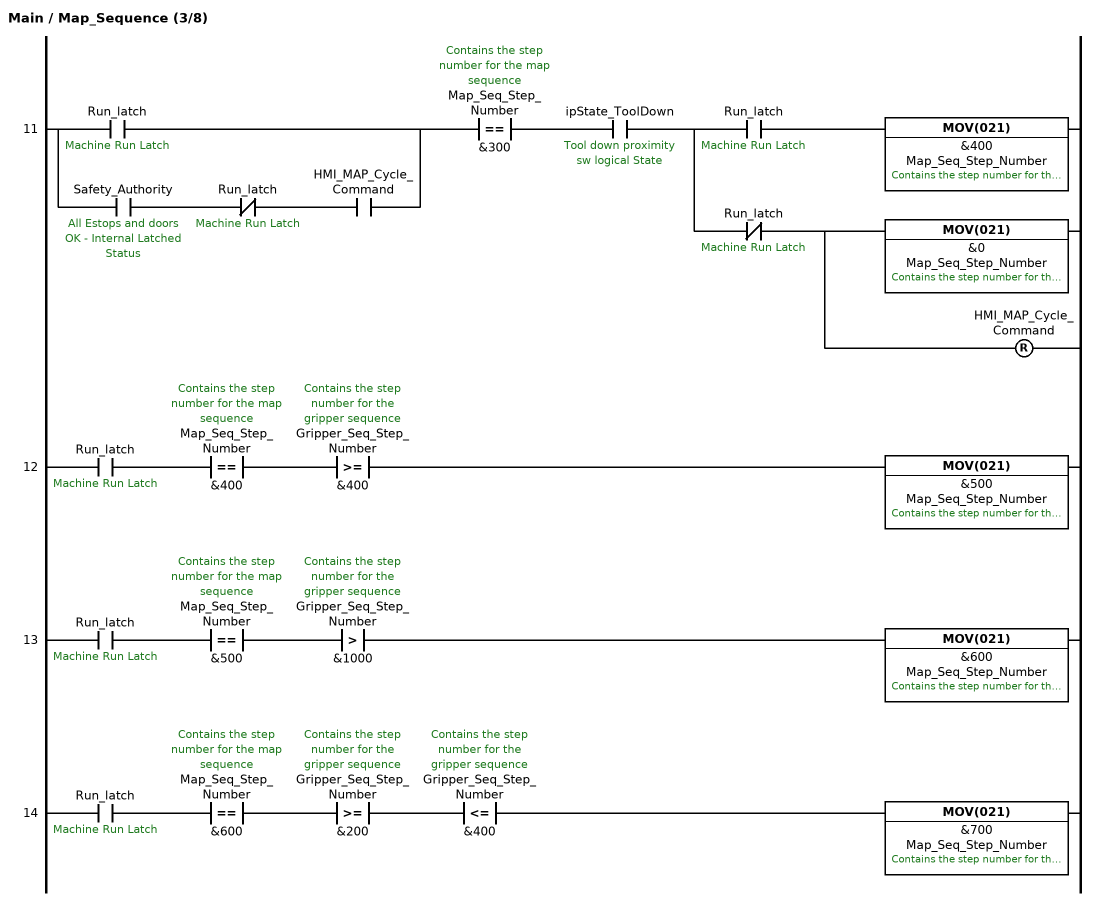
; [picture p48: Main / Map_Sequence, rungs 11-14]
; rung 11
LD Run_latch  ; Machine Run Latch
LD Safety_Authority  ; All Estops and doors OK - Internal Latched Status
ANDNOT Run_latch  ; Machine Run Latch
AND HMI_MAP_Cycle_Command
ORLD
AND=(300) Map_Seq_Step_Number &300  ; Contains the step number for the map sequence
AND ipState_ToolDown  ; Tool down proximity sw logical State
OUT TR0
AND Run_latch  ; Machine Run Latch
MOV(021) &400 Map_Seq_Step_Number  ; Contains the step number for the map sequence
LD TR0
ANDNOT Run_latch  ; Machine Run Latch
MOV(021) &0 Map_Seq_Step_Number  ; Contains the step number for the map sequence
RSET HMI_MAP_Cycle_Command
; rung 12
LD Run_latch  ; Machine Run Latch
AND=(300) Map_Seq_Step_Number &400  ; Contains the step number for the map sequence
AND>=(325) Gripper_Seq_Step_Number &400  ; Contains the step number for the gripper sequence
MOV(021) &500 Map_Seq_Step_Number  ; Contains the step number for the map sequence
; rung 13
LD Run_latch  ; Machine Run Latch
AND=(300) Map_Seq_Step_Number &500  ; Contains the step number for the map sequence
AND>(320) Gripper_Seq_Step_Number &1000  ; Contains the step number for the gripper sequence
MOV(021) &600 Map_Seq_Step_Number  ; Contains the step number for the map sequence
; rung 14
LD Run_latch  ; Machine Run Latch
AND=(300) Map_Seq_Step_Number &600  ; Contains the step number for the map sequence
AND>=(325) Gripper_Seq_Step_Number &200  ; Contains the step number for the gripper sequence
AND<=(315) Gripper_Seq_Step_Number &400  ; Contains the step number for the gripper sequence
MOV(021) &700 Map_Seq_Step_Number  ; Contains the step number for the map sequence

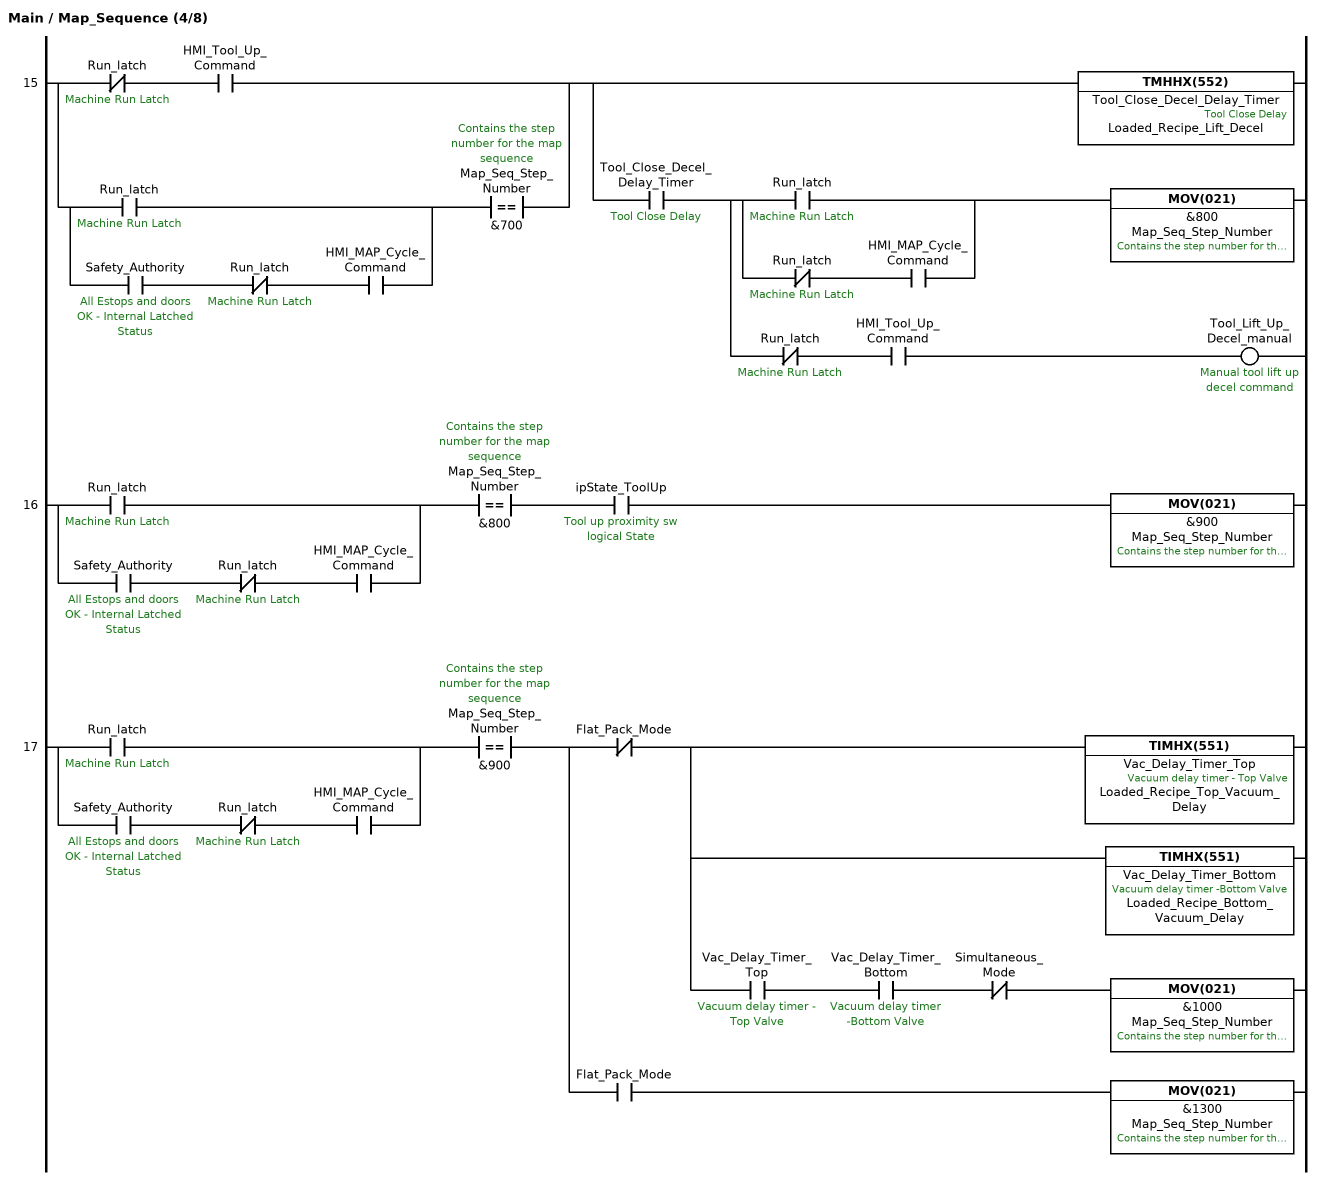
; rung 15
LDNOT Run_latch  ; Machine Run Latch
AND HMI_Tool_Up_Command
LD Run_latch  ; Machine Run Latch
LD Safety_Authority  ; All Estops and doors OK - Internal Latched Status
ANDNOT Run_latch  ; Machine Run Latch
AND HMI_MAP_Cycle_Command
ORLD
AND=(300) Map_Seq_Step_Number &700  ; Contains the step number for the map sequence
ORLD
TMHHX(552) Tool_Close_Decel_Delay_Timer Loaded_Recipe_Lift_Decel  ; Tool Close Delay
AND Tool_Close_Decel_Delay_Timer  ; Tool Close Delay
OUT TR0
LD Run_latch  ; Machine Run Latch
LDNOT Run_latch  ; Machine Run Latch
AND HMI_MAP_Cycle_Command
ORLD
ANDLD
MOV(021) &800 Map_Seq_Step_Number  ; Contains the step number for the map sequence
LD TR0
ANDNOT Run_latch  ; Machine Run Latch
AND HMI_Tool_Up_Command
OUT Tool_Lift_Up_Decel_manual  ; Manual tool lift up decel command
; rung 16
LD Run_latch  ; Machine Run Latch
LD Safety_Authority  ; All Estops and doors OK - Internal Latched Status
ANDNOT Run_latch  ; Machine Run Latch
AND HMI_MAP_Cycle_Command
ORLD
AND=(300) Map_Seq_Step_Number &800  ; Contains the step number for the map sequence
AND ipState_ToolUp  ; Tool up proximity sw logical State
MOV(021) &900 Map_Seq_Step_Number  ; Contains the step number for the map sequence
; rung 17
LD Run_latch  ; Machine Run Latch
LD Safety_Authority  ; All Estops and doors OK - Internal Latched Status
ANDNOT Run_latch  ; Machine Run Latch
AND HMI_MAP_Cycle_Command
ORLD
AND=(300) Map_Seq_Step_Number &900  ; Contains the step number for the map sequence
OUT TR0
ANDNOT Flat_Pack_Mode
TIMHX(551) Vac_Delay_Timer_Top Loaded_Recipe_Top_Vacuum_Delay  ; Vacuum delay timer - Top Valve
TIMHX(551) Vac_Delay_Timer_Bottom Loaded_Recipe_Bottom_Vacuum_Delay  ; Vacuum delay timer -Bottom Valve
AND Vac_Delay_Timer_Top  ; Vacuum delay timer - Top Valve
AND Vac_Delay_Timer_Bottom  ; Vacuum delay timer -Bottom Valve
ANDNOT Simultaneous_Mode
MOV(021) &1000 Map_Seq_Step_Number  ; Contains the step number for the map sequence
LD TR0
AND Flat_Pack_Mode
MOV(021) &1300 Map_Seq_Step_Number  ; Contains the step number for the map sequence

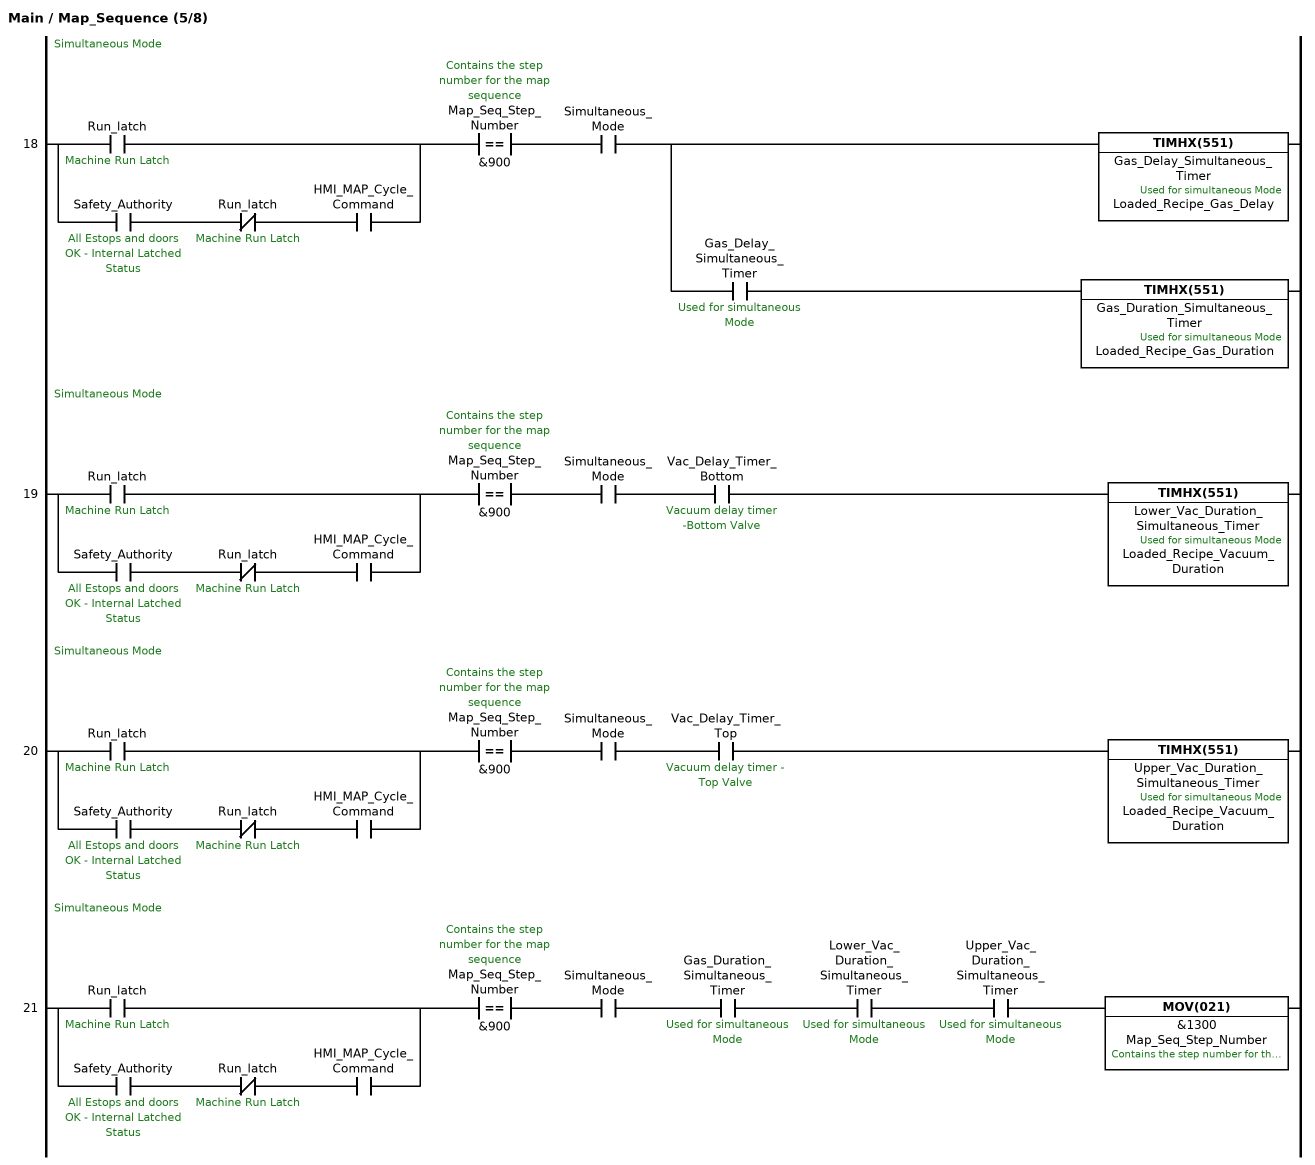
; rung 18: Simultaneous Mode
LD Run_latch  ; Machine Run Latch
LD Safety_Authority  ; All Estops and doors OK - Internal Latched Status
ANDNOT Run_latch  ; Machine Run Latch
AND HMI_MAP_Cycle_Command
ORLD
AND=(300) Map_Seq_Step_Number &900  ; Contains the step number for the map sequence
AND Simultaneous_Mode
TIMHX(551) Gas_Delay_Simultaneous_Timer Loaded_Recipe_Gas_Delay  ; Used for simultaneous Mode
AND Gas_Delay_Simultaneous_Timer  ; Used for simultaneous Mode
TIMHX(551) Gas_Duration_Simultaneous_Timer Loaded_Recipe_Gas_Duration  ; Used for simultaneous Mode
; rung 19: Simultaneous Mode
LD Run_latch  ; Machine Run Latch
LD Safety_Authority  ; All Estops and doors OK - Internal Latched Status
ANDNOT Run_latch  ; Machine Run Latch
AND HMI_MAP_Cycle_Command
ORLD
AND=(300) Map_Seq_Step_Number &900  ; Contains the step number for the map sequence
AND Simultaneous_Mode
AND Vac_Delay_Timer_Bottom  ; Vacuum delay timer -Bottom Valve
TIMHX(551) Lower_Vac_Duration_Simultaneous_Timer Loaded_Recipe_Vacuum_Duration  ; Used for simultaneous Mode
; rung 20: Simultaneous Mode
LD Run_latch  ; Machine Run Latch
LD Safety_Authority  ; All Estops and doors OK - Internal Latched Status
ANDNOT Run_latch  ; Machine Run Latch
AND HMI_MAP_Cycle_Command
ORLD
AND=(300) Map_Seq_Step_Number &900  ; Contains the step number for the map sequence
AND Simultaneous_Mode
AND Vac_Delay_Timer_Top  ; Vacuum delay timer - Top Valve
TIMHX(551) Upper_Vac_Duration_Simultaneous_Timer Loaded_Recipe_Vacuum_Duration  ; Used for simultaneous Mode
; rung 21: Simultaneous Mode
LD Run_latch  ; Machine Run Latch
LD Safety_Authority  ; All Estops and doors OK - Internal Latched Status
ANDNOT Run_latch  ; Machine Run Latch
AND HMI_MAP_Cycle_Command
ORLD
AND=(300) Map_Seq_Step_Number &900  ; Contains the step number for the map sequence
AND Simultaneous_Mode
AND Gas_Duration_Simultaneous_Timer  ; Used for simultaneous Mode
AND Lower_Vac_Duration_Simultaneous_Timer  ; Used for simultaneous Mode
AND Upper_Vac_Duration_Simultaneous_Timer  ; Used for simultaneous Mode
MOV(021) &1300 Map_Seq_Step_Number  ; Contains the step number for the map sequence

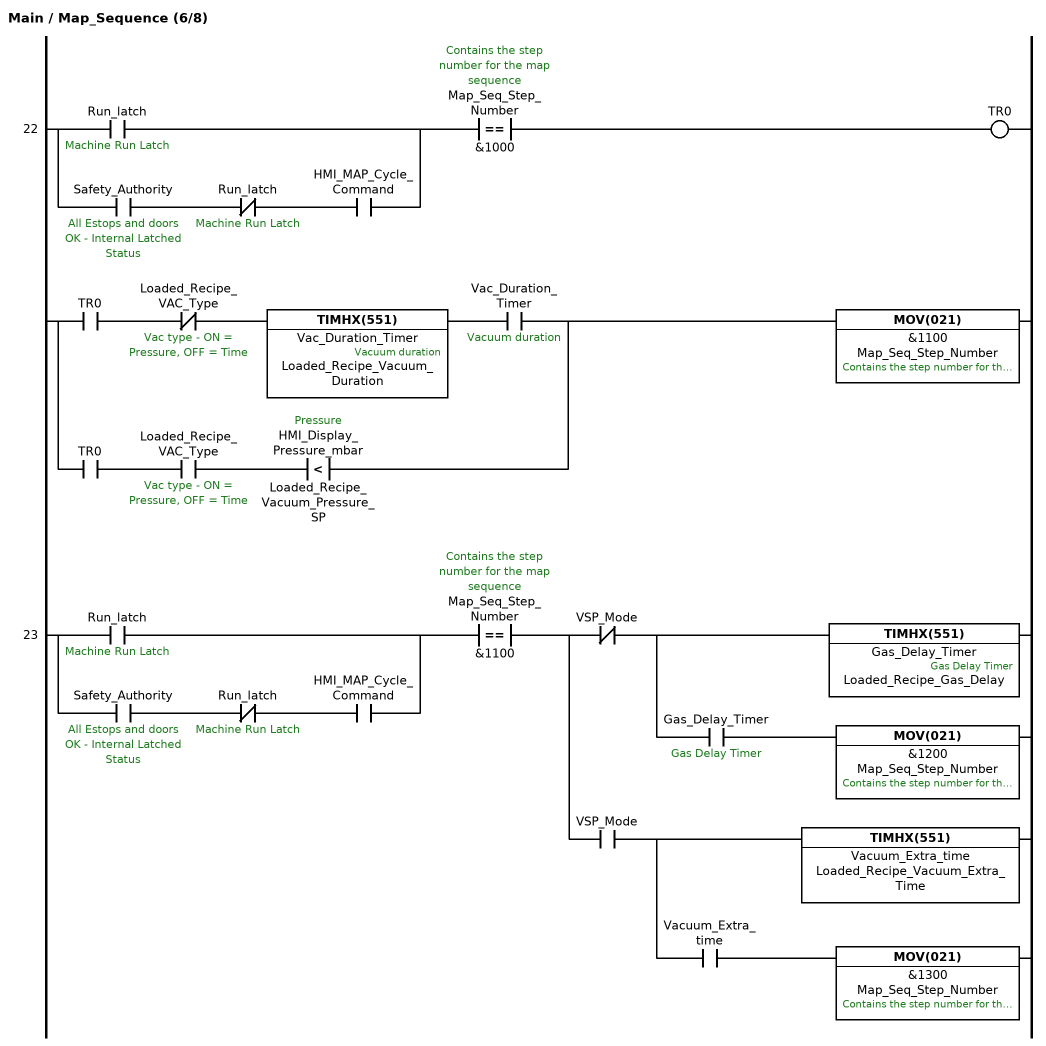
; rung 22
LD Run_latch  ; Machine Run Latch
LD Safety_Authority  ; All Estops and doors OK - Internal Latched Status
ANDNOT Run_latch  ; Machine Run Latch
AND HMI_MAP_Cycle_Command
ORLD
AND=(300) Map_Seq_Step_Number &1000  ; Contains the step number for the map sequence
OUT TR0
ANDNOT Loaded_Recipe_VAC_Type  ; Vac type - ON = Pressure, OFF = Time
TIMHX(551) Vac_Duration_Timer Loaded_Recipe_Vacuum_Duration  ; Vacuum duration
AND Vac_Duration_Timer  ; Vacuum duration
LD TR0
AND Loaded_Recipe_VAC_Type  ; Vac type - ON = Pressure, OFF = Time
AND<(310) HMI_Display_Pressure_mbar Loaded_Recipe_Vacuum_Pressure_SP  ; Pressure
ORLD
MOV(021) &1100 Map_Seq_Step_Number  ; Contains the step number for the map sequence
; rung 23
LD Run_latch  ; Machine Run Latch
LD Safety_Authority  ; All Estops and doors OK - Internal Latched Status
ANDNOT Run_latch  ; Machine Run Latch
AND HMI_MAP_Cycle_Command
ORLD
AND=(300) Map_Seq_Step_Number &1100  ; Contains the step number for the map sequence
OUT TR0
ANDNOT VSP_Mode
TIMHX(551) Gas_Delay_Timer Loaded_Recipe_Gas_Delay  ; Gas Delay Timer
AND Gas_Delay_Timer  ; Gas Delay Timer
MOV(021) &1200 Map_Seq_Step_Number  ; Contains the step number for the map sequence
LD TR0
AND VSP_Mode
TIMHX(551) Vacuum_Extra_time Loaded_Recipe_Vacuum_Extra_Time
AND Vacuum_Extra_time
MOV(021) &1300 Map_Seq_Step_Number  ; Contains the step number for the map sequence

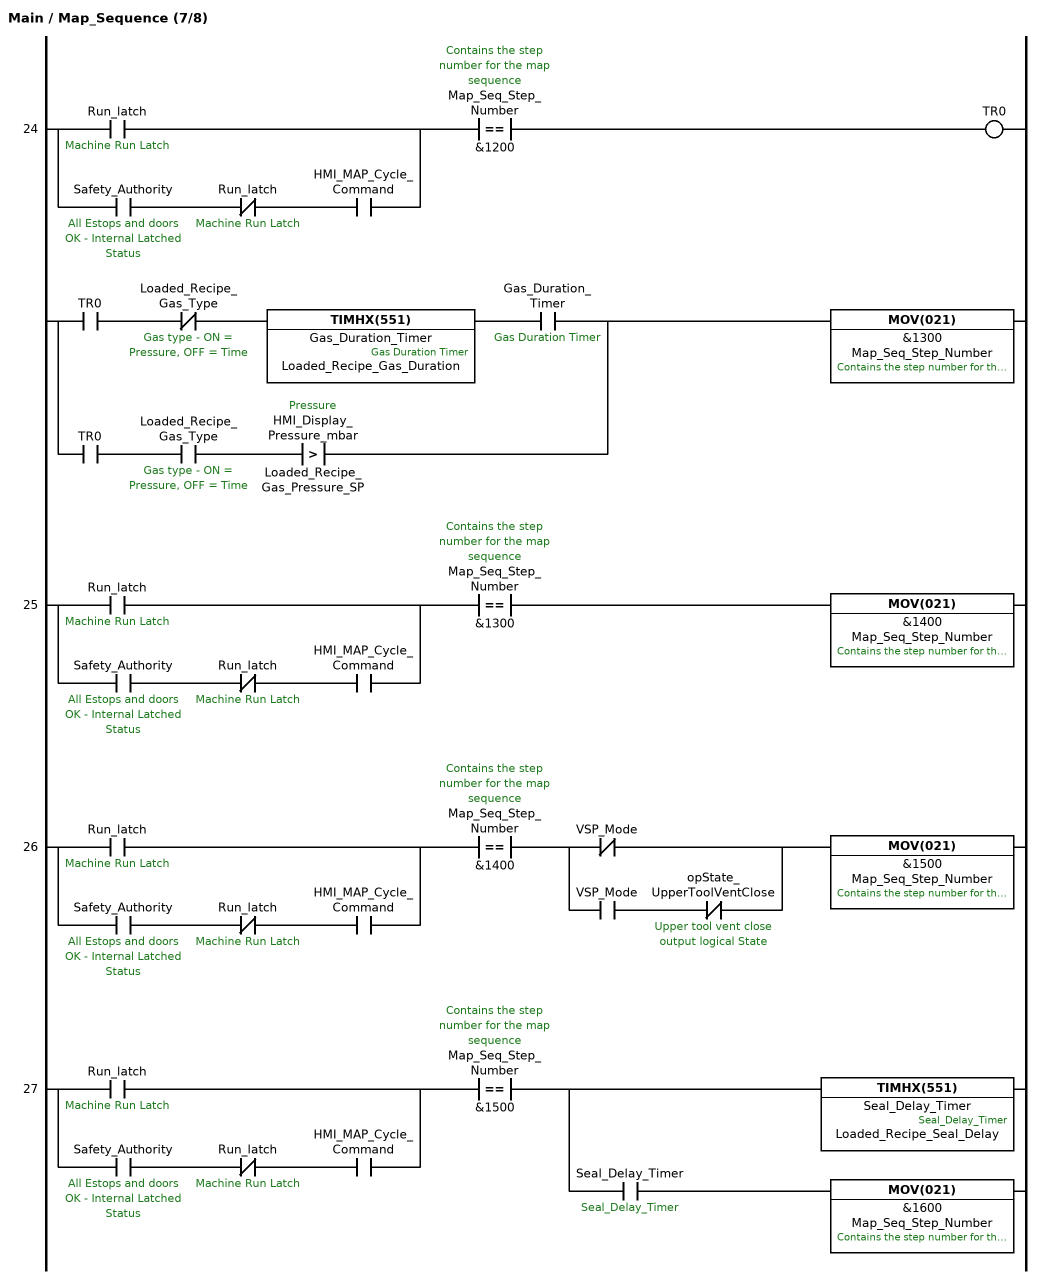
; rung 24
LD Run_latch  ; Machine Run Latch
LD Safety_Authority  ; All Estops and doors OK - Internal Latched Status
ANDNOT Run_latch  ; Machine Run Latch
AND HMI_MAP_Cycle_Command
ORLD
AND=(300) Map_Seq_Step_Number &1200  ; Contains the step number for the map sequence
OUT TR0
ANDNOT Loaded_Recipe_Gas_Type  ; Gas type - ON = Pressure, OFF = Time
TIMHX(551) Gas_Duration_Timer Loaded_Recipe_Gas_Duration  ; Gas Duration Timer
AND Gas_Duration_Timer  ; Gas Duration Timer
LD TR0
AND Loaded_Recipe_Gas_Type  ; Gas type - ON = Pressure, OFF = Time
AND>(320) HMI_Display_Pressure_mbar Loaded_Recipe_Gas_Pressure_SP  ; Pressure
ORLD
MOV(021) &1300 Map_Seq_Step_Number  ; Contains the step number for the map sequence
; rung 25
LD Run_latch  ; Machine Run Latch
LD Safety_Authority  ; All Estops and doors OK - Internal Latched Status
ANDNOT Run_latch  ; Machine Run Latch
AND HMI_MAP_Cycle_Command
ORLD
AND=(300) Map_Seq_Step_Number &1300  ; Contains the step number for the map sequence
MOV(021) &1400 Map_Seq_Step_Number  ; Contains the step number for the map sequence
; rung 26
LD Run_latch  ; Machine Run Latch
LD Safety_Authority  ; All Estops and doors OK - Internal Latched Status
ANDNOT Run_latch  ; Machine Run Latch
AND HMI_MAP_Cycle_Command
ORLD
AND=(300) Map_Seq_Step_Number &1400  ; Contains the step number for the map sequence
LDNOT VSP_Mode
LD VSP_Mode
ANDNOT opState_UpperToolVentClose  ; Upper tool vent close output logical State
ORLD
ANDLD
MOV(021) &1500 Map_Seq_Step_Number  ; Contains the step number for the map sequence
; rung 27
LD Run_latch  ; Machine Run Latch
LD Safety_Authority  ; All Estops and doors OK - Internal Latched Status
ANDNOT Run_latch  ; Machine Run Latch
AND HMI_MAP_Cycle_Command
ORLD
AND=(300) Map_Seq_Step_Number &1500  ; Contains the step number for the map sequence
TIMHX(551) Seal_Delay_Timer Loaded_Recipe_Seal_Delay  ; Seal_Delay_Timer
AND Seal_Delay_Timer  ; Seal_Delay_Timer
MOV(021) &1600 Map_Seq_Step_Number  ; Contains the step number for the map sequence

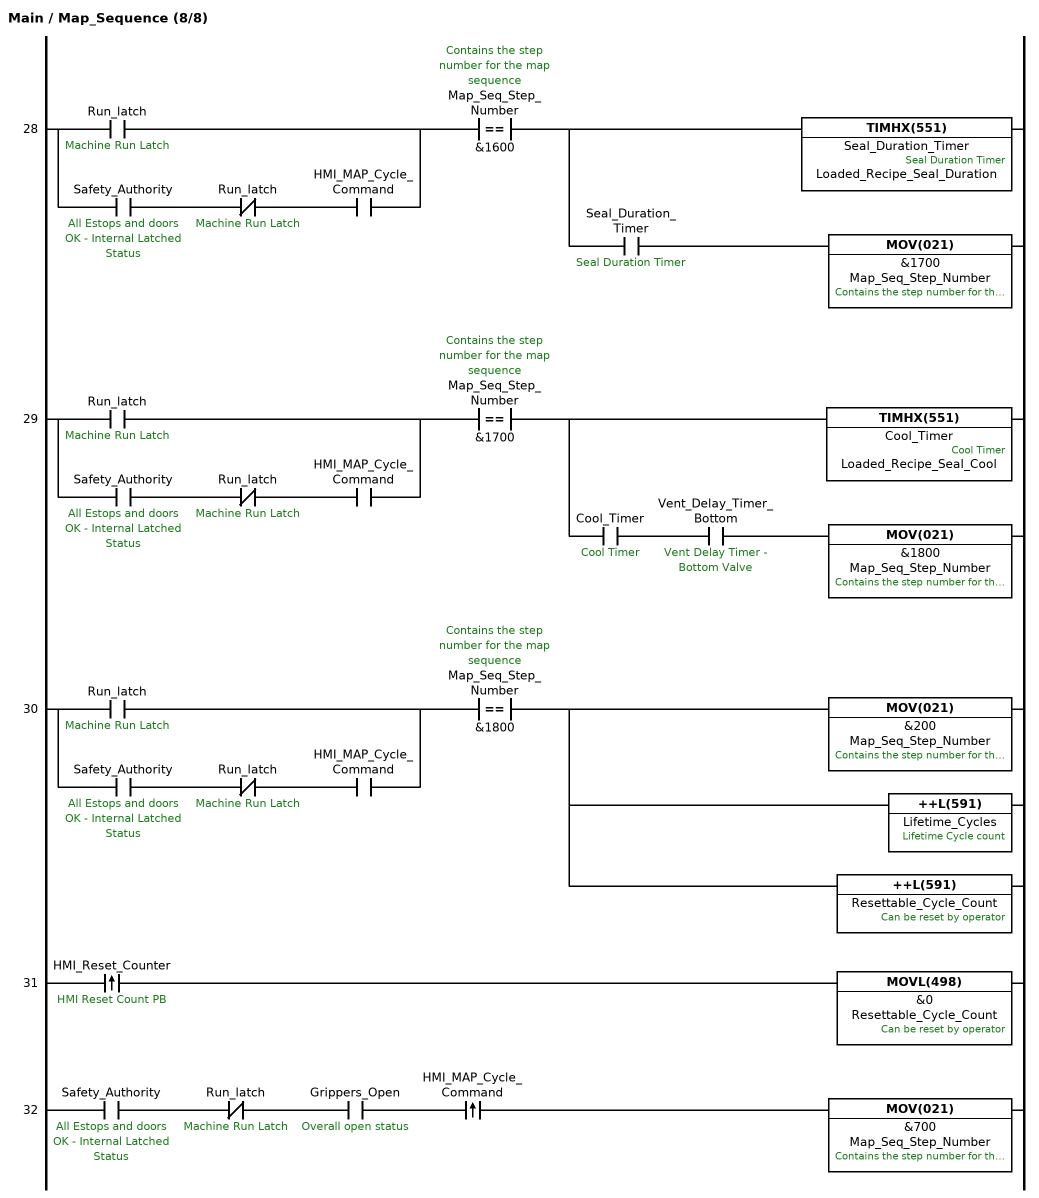
; rung 28
LD Run_latch  ; Machine Run Latch
LD Safety_Authority  ; All Estops and doors OK - Internal Latched Status
ANDNOT Run_latch  ; Machine Run Latch
AND HMI_MAP_Cycle_Command
ORLD
AND=(300) Map_Seq_Step_Number &1600  ; Contains the step number for the map sequence
TIMHX(551) Seal_Duration_Timer Loaded_Recipe_Seal_Duration  ; Seal Duration Timer
AND Seal_Duration_Timer  ; Seal Duration Timer
MOV(021) &1700 Map_Seq_Step_Number  ; Contains the step number for the map sequence
; rung 29
LD Run_latch  ; Machine Run Latch
LD Safety_Authority  ; All Estops and doors OK - Internal Latched Status
ANDNOT Run_latch  ; Machine Run Latch
AND HMI_MAP_Cycle_Command
ORLD
AND=(300) Map_Seq_Step_Number &1700  ; Contains the step number for the map sequence
TIMHX(551) Cool_Timer Loaded_Recipe_Seal_Cool  ; Cool Timer
AND Cool_Timer  ; Cool Timer
AND Vent_Delay_Timer_Bottom  ; Vent Delay Timer - Bottom Valve
MOV(021) &1800 Map_Seq_Step_Number  ; Contains the step number for the map sequence
; rung 30
LD Run_latch  ; Machine Run Latch
LD Safety_Authority  ; All Estops and doors OK - Internal Latched Status
ANDNOT Run_latch  ; Machine Run Latch
AND HMI_MAP_Cycle_Command
ORLD
AND=(300) Map_Seq_Step_Number &1800  ; Contains the step number for the map sequence
MOV(021) &200 Map_Seq_Step_Number  ; Contains the step number for the map sequence
++L(591) Lifetime_Cycles  ; Lifetime Cycle count
++L(591) Resettable_Cycle_Count  ; Can be reset by operator
; rung 31
@LD HMI_Reset_Counter  ; HMI Reset Count PB
MOVL(498) &0 Resettable_Cycle_Count  ; Can be reset by operator
; rung 32
LD Safety_Authority  ; All Estops and doors OK - Internal Latched Status
ANDNOT Run_latch  ; Machine Run Latch
AND Grippers_Open  ; Overall open status
@AND HMI_MAP_Cycle_Command
MOV(021) &700 Map_Seq_Step_Number  ; Contains the step number for the map sequence

### Section Map_Outputs

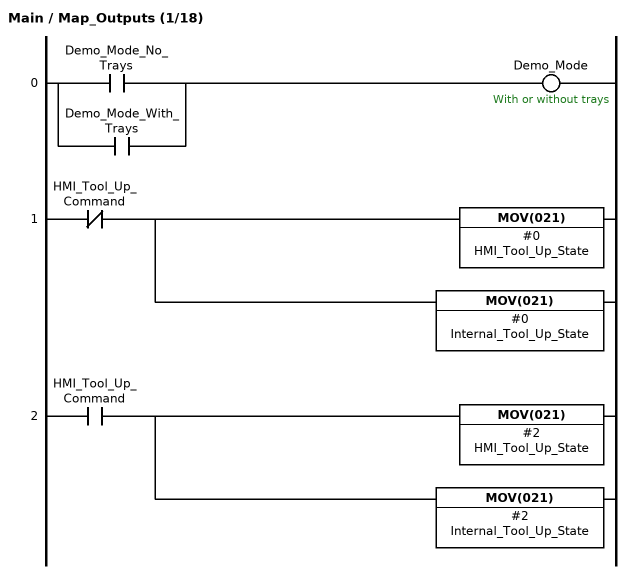
; rung 0
LD Demo_Mode_No_Trays
OR Demo_Mode_With_Trays
OUT Demo_Mode  ; With or without trays
; rung 1
LDNOT HMI_Tool_Up_Command
MOV(021) #0 HMI_Tool_Up_State
MOV(021) #0 Internal_Tool_Up_State
; rung 2
LD HMI_Tool_Up_Command
MOV(021) #2 HMI_Tool_Up_State
MOV(021) #2 Internal_Tool_Up_State

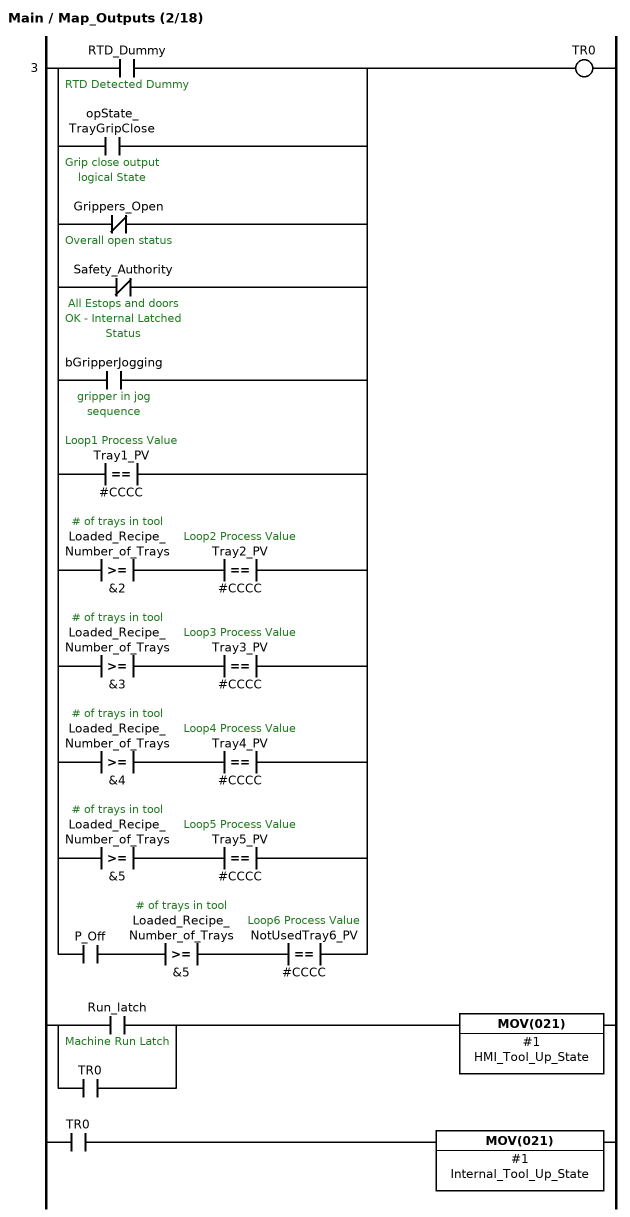
; rung 3
LD Run_latch  ; Machine Run Latch
LD RTD_Dummy  ; RTD Detected Dummy
OR opState_TrayGripClose  ; Grip close output logical State
ORNOT Grippers_Open  ; Overall open status
ORNOT Safety_Authority  ; All Estops and doors OK - Internal Latched Status
OR bGripperJogging  ; gripper in jog sequence
OR=S(302) Tray1_PV #CCCC  ; Loop1 Process Value
LD>=(325) Loaded_Recipe_Number_of_Trays &2  ; # of trays in tool
AND=S(302) Tray2_PV #CCCC  ; Loop2 Process Value
ORLD
LD>=(325) Loaded_Recipe_Number_of_Trays &3  ; # of trays in tool
AND=S(302) Tray3_PV #CCCC  ; Loop3 Process Value
ORLD
LD>=(325) Loaded_Recipe_Number_of_Trays &4  ; # of trays in tool
AND=S(302) Tray4_PV #CCCC  ; Loop4 Process Value
ORLD
LD>=(325) Loaded_Recipe_Number_of_Trays &5  ; # of trays in tool
AND=S(302) Tray5_PV #CCCC  ; Loop5 Process Value
ORLD
LD P_Off
AND>=(325) Loaded_Recipe_Number_of_Trays &5  ; # of trays in tool
AND=S(302) NotUsedTray6_PV #CCCC  ; Loop6 Process Value
ORLD
OUT TR0
ORLD
MOV(021) #1 HMI_Tool_Up_State
LD TR0
MOV(021) #1 Internal_Tool_Up_State

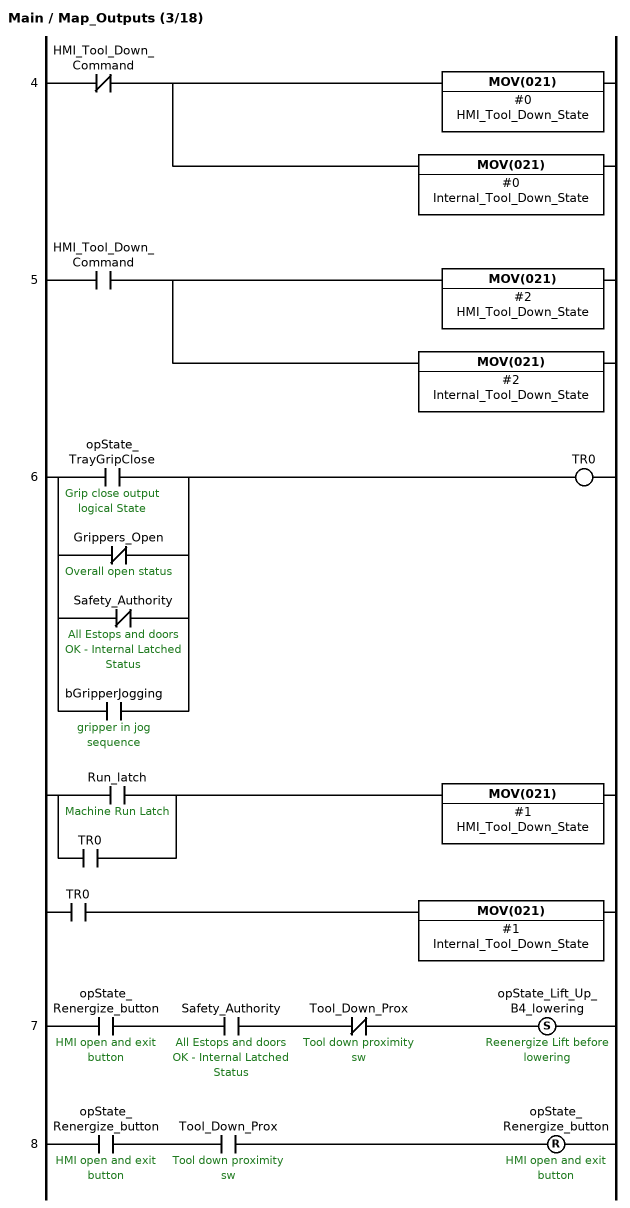
; rung 4
LDNOT HMI_Tool_Down_Command
MOV(021) #0 HMI_Tool_Down_State
MOV(021) #0 Internal_Tool_Down_State
; rung 5
LD HMI_Tool_Down_Command
MOV(021) #2 HMI_Tool_Down_State
MOV(021) #2 Internal_Tool_Down_State
; rung 6
LD Run_latch  ; Machine Run Latch
LD opState_TrayGripClose  ; Grip close output logical State
ORNOT Grippers_Open  ; Overall open status
ORNOT Safety_Authority  ; All Estops and doors OK - Internal Latched Status
OR bGripperJogging  ; gripper in jog sequence
OUT TR0
ORLD
MOV(021) #1 HMI_Tool_Down_State
LD TR0
MOV(021) #1 Internal_Tool_Down_State
; rung 7
LD opState_Renergize_button  ; HMI open and exit button
AND Safety_Authority  ; All Estops and doors OK - Internal Latched Status
ANDNOT Tool_Down_Prox  ; Tool down proximity sw
SET opState_Lift_Up_B4_lowering  ; Reenergize Lift before lowering
; rung 8
LD opState_Renergize_button  ; HMI open and exit button
AND Tool_Down_Prox  ; Tool down proximity sw
RSET opState_Renergize_button  ; HMI open and exit button

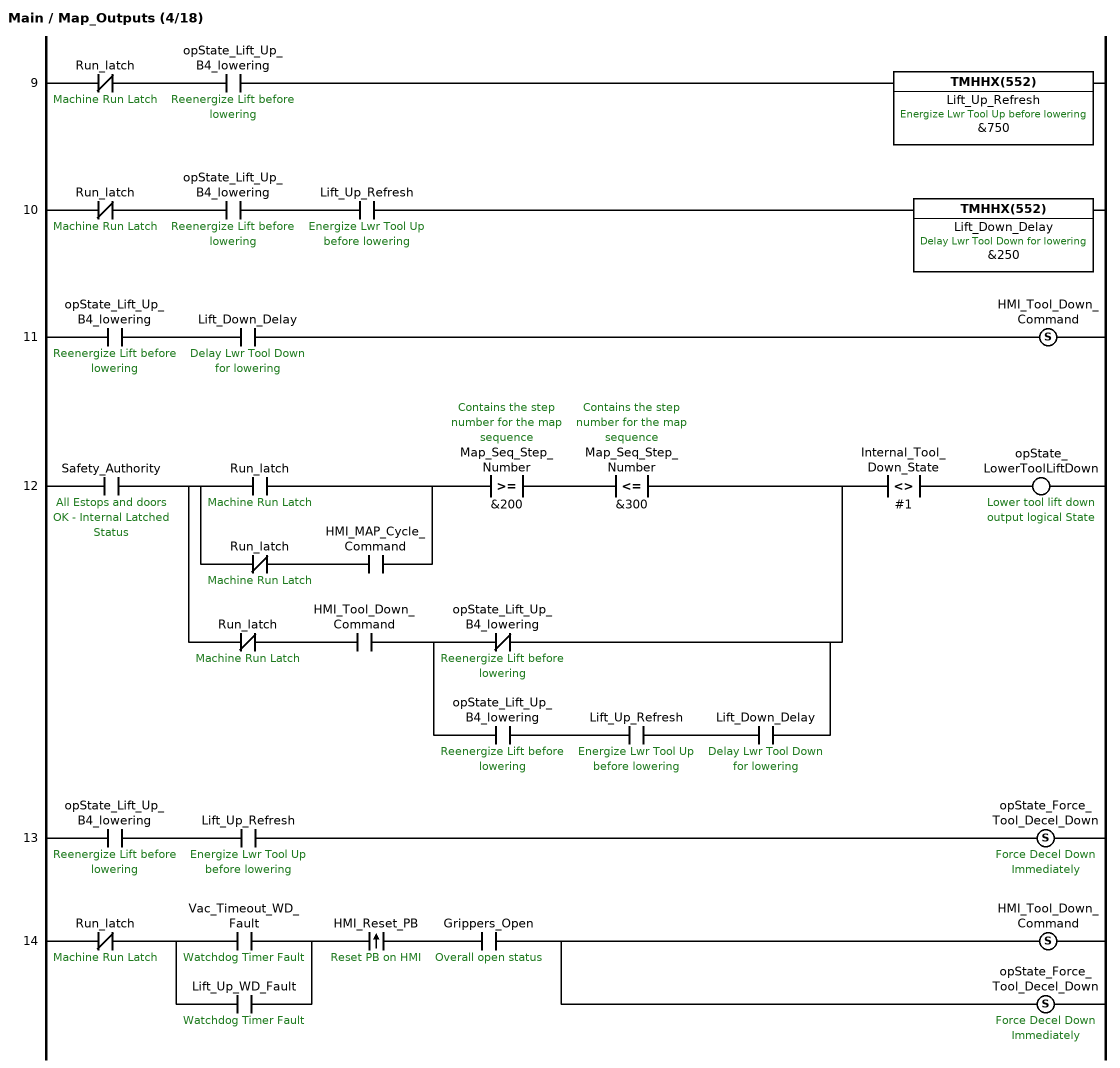
; rung 9
LDNOT Run_latch  ; Machine Run Latch
AND opState_Lift_Up_B4_lowering  ; Reenergize Lift before lowering
TMHHX(552) Lift_Up_Refresh &750  ; Energize Lwr Tool Up before lowering
; rung 10
LDNOT Run_latch  ; Machine Run Latch
AND opState_Lift_Up_B4_lowering  ; Reenergize Lift before lowering
AND Lift_Up_Refresh  ; Energize Lwr Tool Up before lowering
TMHHX(552) Lift_Down_Delay &250  ; Delay Lwr Tool Down for lowering
; rung 11
LD opState_Lift_Up_B4_lowering  ; Reenergize Lift before lowering
AND Lift_Down_Delay  ; Delay Lwr Tool Down for lowering
SET HMI_Tool_Down_Command
; rung 12
LD Safety_Authority  ; All Estops and doors OK - Internal Latched Status
LD Run_latch  ; Machine Run Latch
LDNOT Run_latch  ; Machine Run Latch
AND HMI_MAP_Cycle_Command
ORLD
AND>=(325) Map_Seq_Step_Number &200  ; Contains the step number for the map sequence
AND<=(315) Map_Seq_Step_Number &300  ; Contains the step number for the map sequence
LDNOT Run_latch  ; Machine Run Latch
AND HMI_Tool_Down_Command
LDNOT opState_Lift_Up_B4_lowering  ; Reenergize Lift before lowering
LD opState_Lift_Up_B4_lowering  ; Reenergize Lift before lowering
AND Lift_Up_Refresh  ; Energize Lwr Tool Up before lowering
AND Lift_Down_Delay  ; Delay Lwr Tool Down for lowering
ORLD
ANDLD
ORLD
ANDLD
AND<>(305) Internal_Tool_Down_State #1
OUT opState_LowerToolLiftDown  ; Lower tool lift down output logical State
; rung 13
LD opState_Lift_Up_B4_lowering  ; Reenergize Lift before lowering
AND Lift_Up_Refresh  ; Energize Lwr Tool Up before lowering
SET opState_Force_Tool_Decel_Down  ; Force Decel Down Immediately
; rung 14
LDNOT Run_latch  ; Machine Run Latch
LD Vac_Timeout_WD_Fault  ; Watchdog Timer Fault
OR Lift_Up_WD_Fault  ; Watchdog Timer Fault
ANDLD
@AND HMI_Reset_PB  ; Reset PB on HMI
AND Grippers_Open  ; Overall open status
SET HMI_Tool_Down_Command
SET opState_Force_Tool_Decel_Down  ; Force Decel Down Immediately

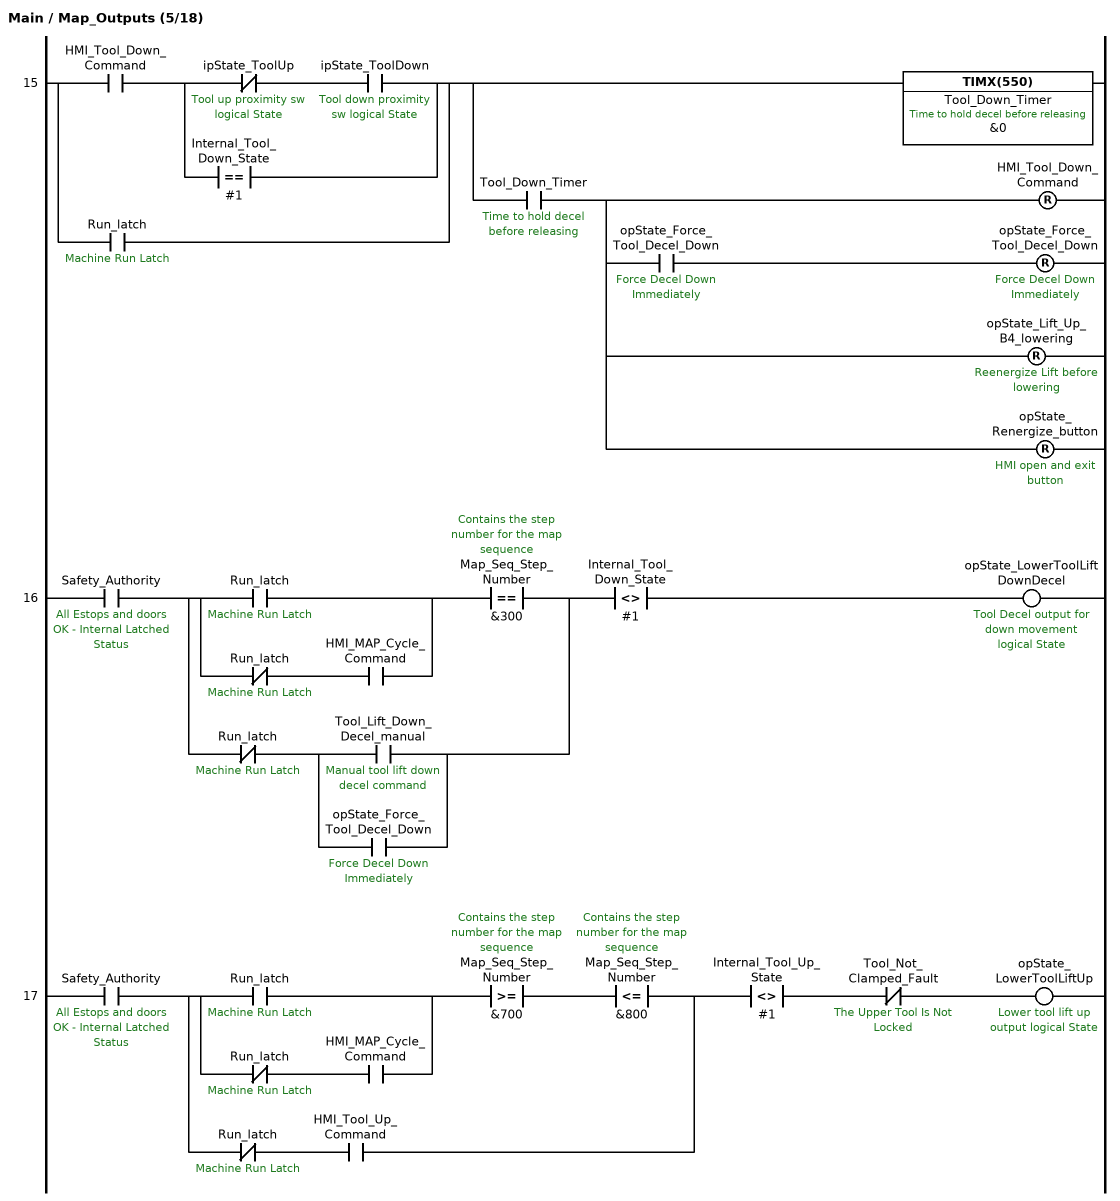
; rung 15
LD HMI_Tool_Down_Command
LDNOT ipState_ToolUp  ; Tool up proximity sw logical State
AND ipState_ToolDown  ; Tool down proximity sw logical State
OR=(300) Internal_Tool_Down_State #1
ANDLD
OR Run_latch  ; Machine Run Latch
TIMX(550) Tool_Down_Timer &0  ; Time to hold decel before releasing
AND Tool_Down_Timer  ; Time to hold decel before releasing
OUT TR0
RSET HMI_Tool_Down_Command
AND opState_Force_Tool_Decel_Down  ; Force Decel Down Immediately
RSET opState_Force_Tool_Decel_Down  ; Force Decel Down Immediately
LD TR0
RSET opState_Lift_Up_B4_lowering  ; Reenergize Lift before lowering
RSET opState_Renergize_button  ; HMI open and exit button
; rung 16
LD Safety_Authority  ; All Estops and doors OK - Internal Latched Status
LD Run_latch  ; Machine Run Latch
LDNOT Run_latch  ; Machine Run Latch
AND HMI_MAP_Cycle_Command
ORLD
AND=(300) Map_Seq_Step_Number &300  ; Contains the step number for the map sequence
LDNOT Run_latch  ; Machine Run Latch
LD Tool_Lift_Down_Decel_manual  ; Manual tool lift down decel command
OR opState_Force_Tool_Decel_Down  ; Force Decel Down Immediately
ANDLD
ORLD
ANDLD
AND<>(305) Internal_Tool_Down_State #1
OUT opState_LowerToolLiftDownDecel  ; Tool Decel output for down movement logical State
; rung 17
LD Safety_Authority  ; All Estops and doors OK - Internal Latched Status
LD Run_latch  ; Machine Run Latch
LDNOT Run_latch  ; Machine Run Latch
AND HMI_MAP_Cycle_Command
ORLD
AND>=(325) Map_Seq_Step_Number &700  ; Contains the step number for the map sequence
AND<=(315) Map_Seq_Step_Number &800  ; Contains the step number for the map sequence
LDNOT Run_latch  ; Machine Run Latch
AND HMI_Tool_Up_Command
ORLD
ANDLD
AND<>(305) Internal_Tool_Up_State #1
ANDNOT Tool_Not_Clamped_Fault  ; The Upper Tool Is Not Locked
OUT opState_LowerToolLiftUp  ; Lower tool lift up output logical State

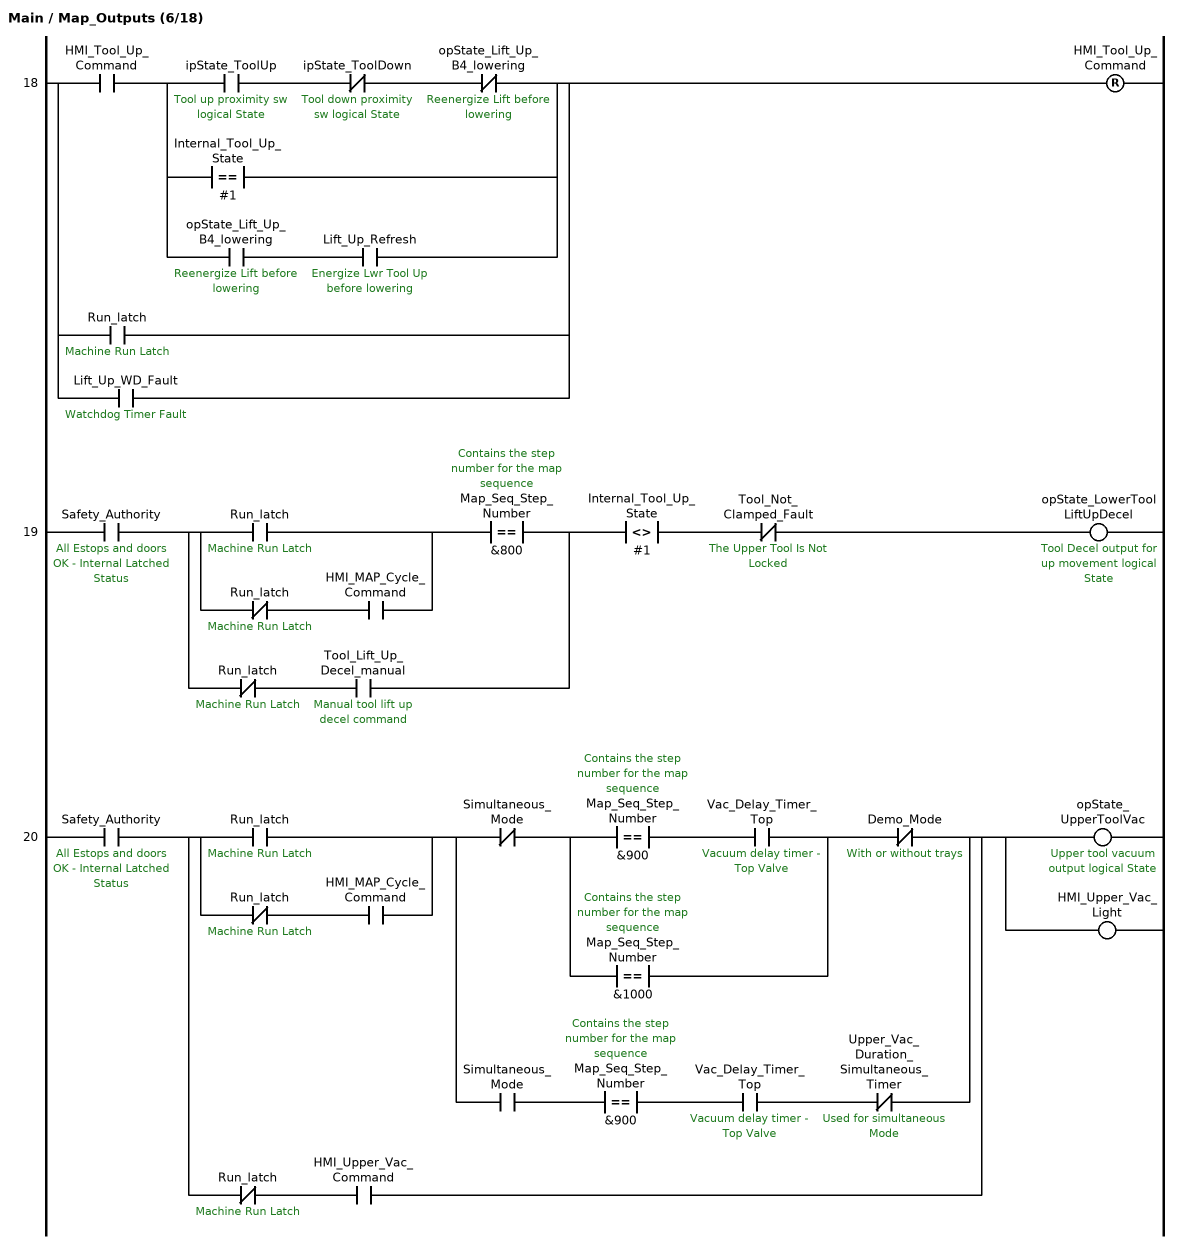
; rung 18
LD HMI_Tool_Up_Command
LD ipState_ToolUp  ; Tool up proximity sw logical State
ANDNOT ipState_ToolDown  ; Tool down proximity sw logical State
ANDNOT opState_Lift_Up_B4_lowering  ; Reenergize Lift before lowering
OR=(300) Internal_Tool_Up_State #1
LD opState_Lift_Up_B4_lowering  ; Reenergize Lift before lowering
AND Lift_Up_Refresh  ; Energize Lwr Tool Up before lowering
ORLD
ANDLD
OR Run_latch  ; Machine Run Latch
OR Lift_Up_WD_Fault  ; Watchdog Timer Fault
RSET HMI_Tool_Up_Command
; rung 19
LD Safety_Authority  ; All Estops and doors OK - Internal Latched Status
LD Run_latch  ; Machine Run Latch
LDNOT Run_latch  ; Machine Run Latch
AND HMI_MAP_Cycle_Command
ORLD
AND=(300) Map_Seq_Step_Number &800  ; Contains the step number for the map sequence
LDNOT Run_latch  ; Machine Run Latch
AND Tool_Lift_Up_Decel_manual  ; Manual tool lift up decel command
ORLD
ANDLD
AND<>(305) Internal_Tool_Up_State #1
ANDNOT Tool_Not_Clamped_Fault  ; The Upper Tool Is Not Locked
OUT opState_LowerToolLiftUpDecel  ; Tool Decel output for up movement logical State
; rung 20
LD Safety_Authority  ; All Estops and doors OK - Internal Latched Status
LD Run_latch  ; Machine Run Latch
LDNOT Run_latch  ; Machine Run Latch
AND HMI_MAP_Cycle_Command
ORLD
LDNOT Simultaneous_Mode
LD=(300) Map_Seq_Step_Number &900  ; Contains the step number for the map sequence
AND Vac_Delay_Timer_Top  ; Vacuum delay timer - Top Valve
OR=(300) Map_Seq_Step_Number &1000  ; Contains the step number for the map sequence
ANDLD
ANDNOT Demo_Mode  ; With or without trays
LD Simultaneous_Mode
AND=(300) Map_Seq_Step_Number &900  ; Contains the step number for the map sequence
AND Vac_Delay_Timer_Top  ; Vacuum delay timer - Top Valve
ANDNOT Upper_Vac_Duration_Simultaneous_Timer  ; Used for simultaneous Mode
ORLD
ANDLD
LDNOT Run_latch  ; Machine Run Latch
AND HMI_Upper_Vac_Command
ORLD
ANDLD
OUT opState_UpperToolVac  ; Upper tool vacuum output logical State
OUT HMI_Upper_Vac_Light

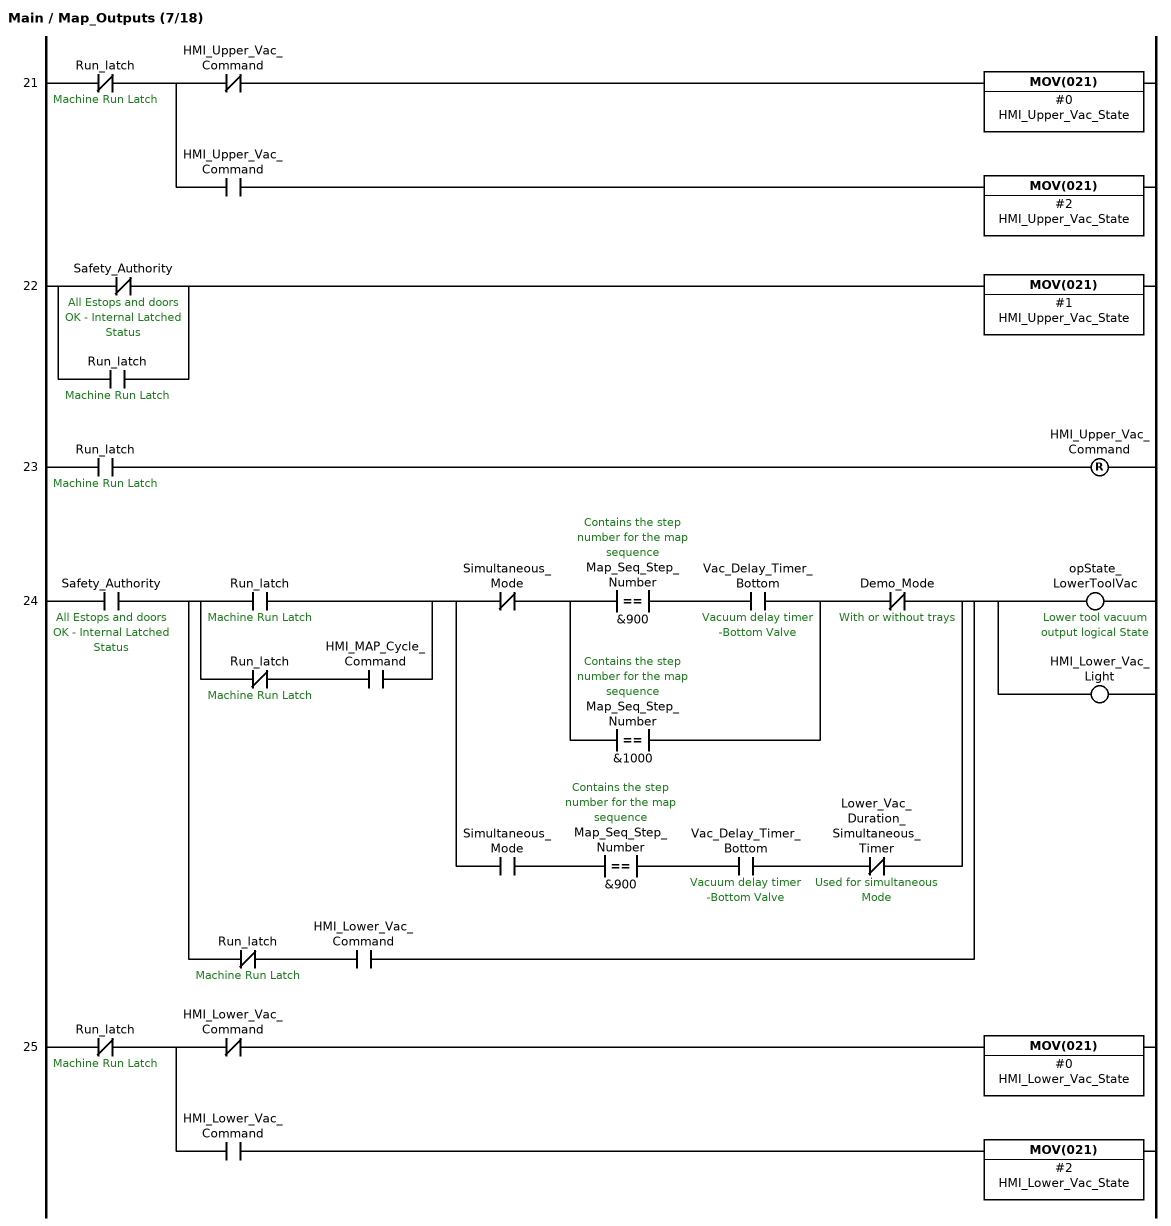
; rung 21
LDNOT Run_latch  ; Machine Run Latch
OUT TR0
ANDNOT HMI_Upper_Vac_Command
MOV(021) #0 HMI_Upper_Vac_State
LD TR0
AND HMI_Upper_Vac_Command
MOV(021) #2 HMI_Upper_Vac_State
; rung 22
LDNOT Safety_Authority  ; All Estops and doors OK - Internal Latched Status
OR Run_latch  ; Machine Run Latch
MOV(021) #1 HMI_Upper_Vac_State
; rung 23
LD Run_latch  ; Machine Run Latch
RSET HMI_Upper_Vac_Command
; rung 24
LD Safety_Authority  ; All Estops and doors OK - Internal Latched Status
LD Run_latch  ; Machine Run Latch
LDNOT Run_latch  ; Machine Run Latch
AND HMI_MAP_Cycle_Command
ORLD
LDNOT Simultaneous_Mode
LD=(300) Map_Seq_Step_Number &900  ; Contains the step number for the map sequence
AND Vac_Delay_Timer_Bottom  ; Vacuum delay timer -Bottom Valve
OR=(300) Map_Seq_Step_Number &1000  ; Contains the step number for the map sequence
ANDLD
ANDNOT Demo_Mode  ; With or without trays
LD Simultaneous_Mode
AND=(300) Map_Seq_Step_Number &900  ; Contains the step number for the map sequence
AND Vac_Delay_Timer_Bottom  ; Vacuum delay timer -Bottom Valve
ANDNOT Lower_Vac_Duration_Simultaneous_Timer  ; Used for simultaneous Mode
ORLD
ANDLD
LDNOT Run_latch  ; Machine Run Latch
AND HMI_Lower_Vac_Command
ORLD
ANDLD
OUT opState_LowerToolVac  ; Lower tool vacuum output logical State
OUT HMI_Lower_Vac_Light
; rung 25
LDNOT Run_latch  ; Machine Run Latch
OUT TR0
ANDNOT HMI_Lower_Vac_Command
MOV(021) #0 HMI_Lower_Vac_State
LD TR0
AND HMI_Lower_Vac_Command
MOV(021) #2 HMI_Lower_Vac_State

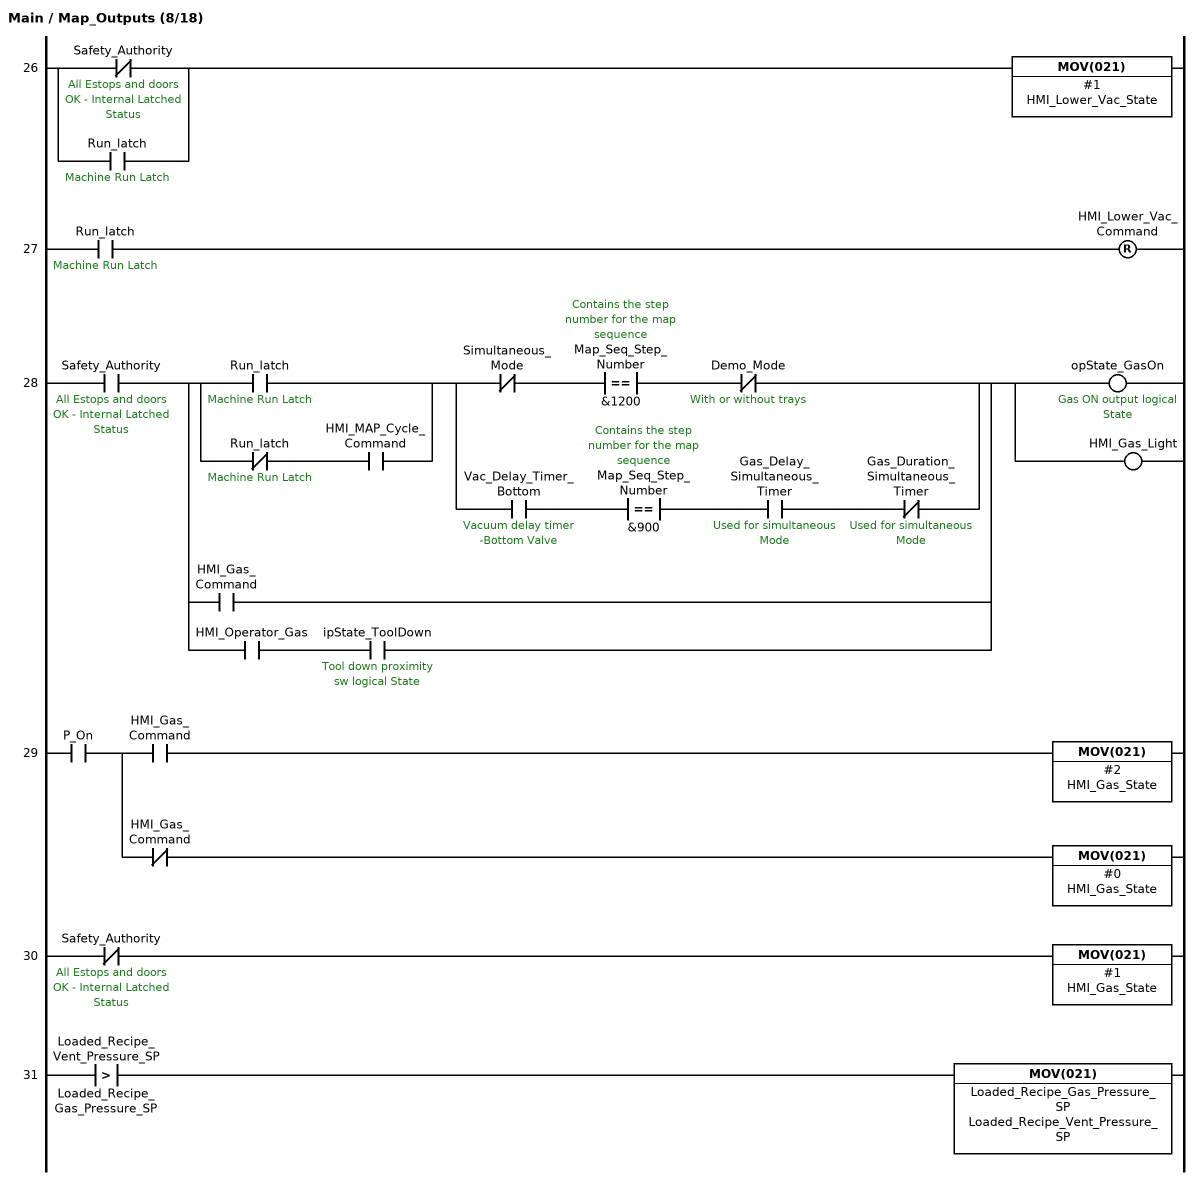
; rung 26
LDNOT Safety_Authority  ; All Estops and doors OK - Internal Latched Status
OR Run_latch  ; Machine Run Latch
MOV(021) #1 HMI_Lower_Vac_State
; rung 27
LD Run_latch  ; Machine Run Latch
RSET HMI_Lower_Vac_Command
; rung 28
LD Safety_Authority  ; All Estops and doors OK - Internal Latched Status
LD Run_latch  ; Machine Run Latch
LDNOT Run_latch  ; Machine Run Latch
AND HMI_MAP_Cycle_Command
ORLD
LDNOT Simultaneous_Mode
AND=(300) Map_Seq_Step_Number &1200  ; Contains the step number for the map sequence
ANDNOT Demo_Mode  ; With or without trays
LD Vac_Delay_Timer_Bottom  ; Vacuum delay timer -Bottom Valve
AND=(300) Map_Seq_Step_Number &900  ; Contains the step number for the map sequence
AND Gas_Delay_Simultaneous_Timer  ; Used for simultaneous Mode
ANDNOT Gas_Duration_Simultaneous_Timer  ; Used for simultaneous Mode
ORLD
ANDLD
OR HMI_Gas_Command
LD HMI_Operator_Gas
AND ipState_ToolDown  ; Tool down proximity sw logical State
ORLD
ANDLD
OUT opState_GasOn  ; Gas ON output logical State
OUT HMI_Gas_Light
; rung 29
LD P_On
OUT TR0
AND HMI_Gas_Command
MOV(021) #2 HMI_Gas_State
LD TR0
ANDNOT HMI_Gas_Command
MOV(021) #0 HMI_Gas_State
; rung 30
LDNOT Safety_Authority  ; All Estops and doors OK - Internal Latched Status
MOV(021) #1 HMI_Gas_State
; rung 31
LD>(320) Loaded_Recipe_Vent_Pressure_SP Loaded_Recipe_Gas_Pressure_SP
MOV(021) Loaded_Recipe_Gas_Pressure_SP Loaded_Recipe_Vent_Pressure_SP

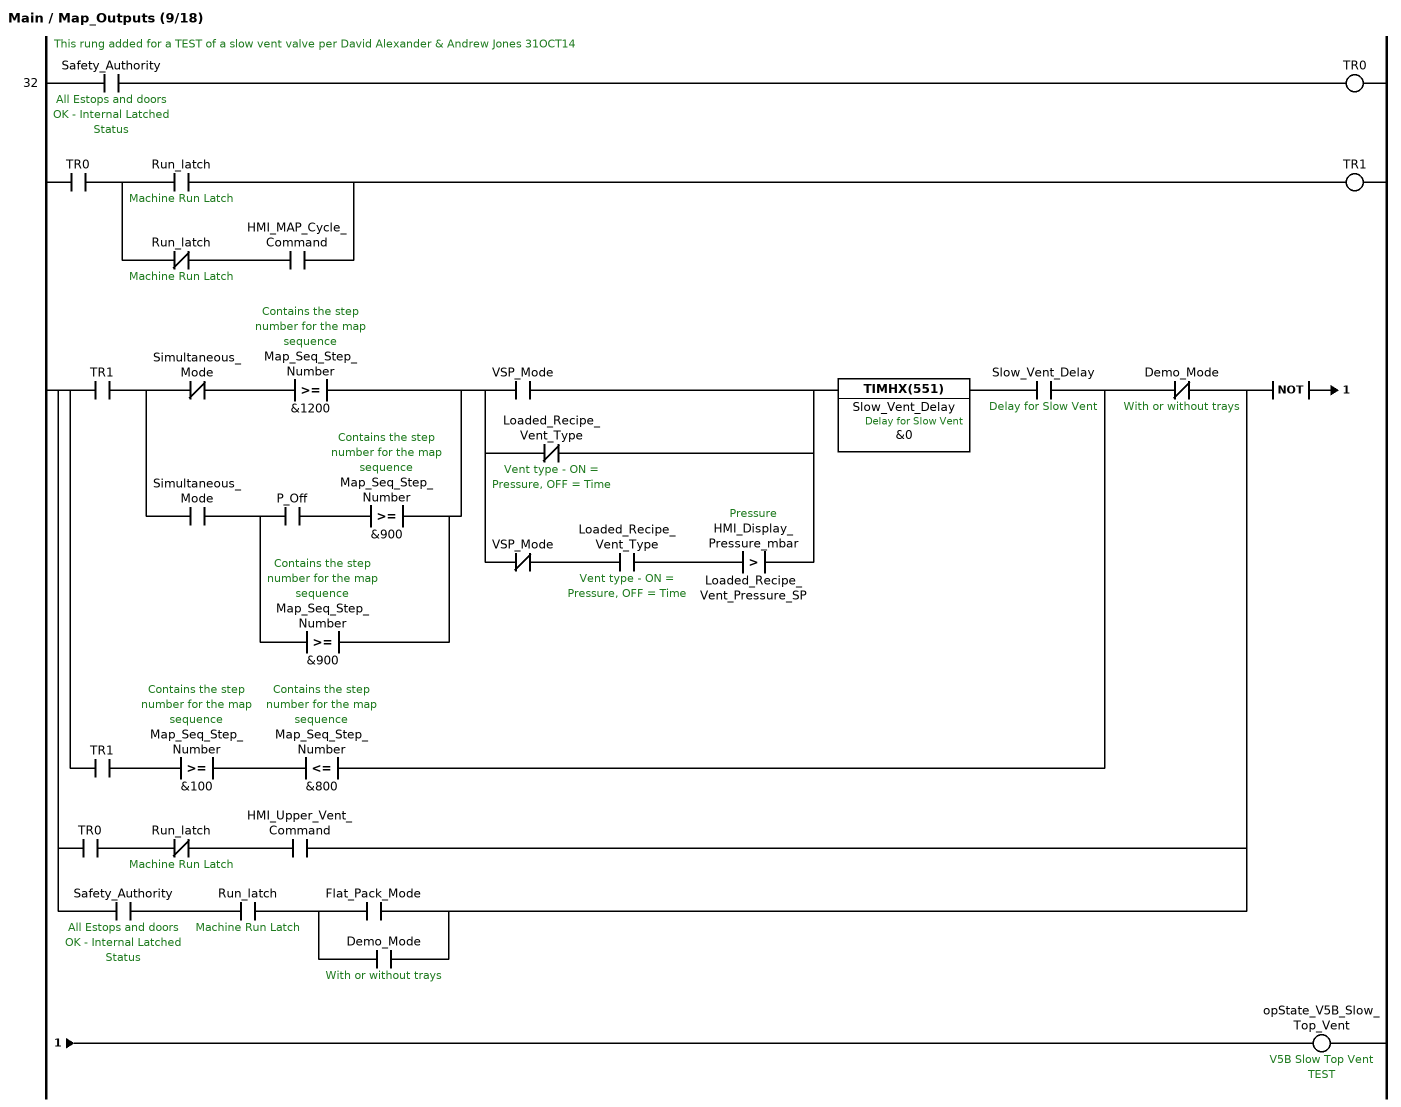
; rung 32: This rung added for a TEST of a slow vent valve per David Alexander & Andrew Jones 31OCT14
LD Safety_Authority  ; All Estops and doors OK - Internal Latched Status
OUT TR0
LD Run_latch  ; Machine Run Latch
LDNOT Run_latch  ; Machine Run Latch
AND HMI_MAP_Cycle_Command
ORLD
ANDLD
OUT TR1
LDNOT Simultaneous_Mode
AND>=(325) Map_Seq_Step_Number &1200  ; Contains the step number for the map sequence
LD Simultaneous_Mode
LD P_Off
AND>=(325) Map_Seq_Step_Number &900  ; Contains the step number for the map sequence
OR>=(325) Map_Seq_Step_Number &900  ; Contains the step number for the map sequence
ANDLD
ORLD
ANDLD
LD VSP_Mode
ORNOT Loaded_Recipe_Vent_Type  ; Vent type - ON = Pressure, OFF = Time
LDNOT VSP_Mode
AND Loaded_Recipe_Vent_Type  ; Vent type - ON = Pressure, OFF = Time
AND>(320) HMI_Display_Pressure_mbar Loaded_Recipe_Vent_Pressure_SP  ; Pressure
ORLD
ANDLD
TIMHX(551) Slow_Vent_Delay &0  ; Delay for Slow Vent
AND Slow_Vent_Delay  ; Delay for Slow Vent
LD TR1
AND>=(325) Map_Seq_Step_Number &100  ; Contains the step number for the map sequence
AND<=(315) Map_Seq_Step_Number &800  ; Contains the step number for the map sequence
ORLD
ANDNOT Demo_Mode  ; With or without trays
LD TR0
ANDNOT Run_latch  ; Machine Run Latch
AND HMI_Upper_Vent_Command
LD Safety_Authority  ; All Estops and doors OK - Internal Latched Status
AND Run_latch  ; Machine Run Latch
LD Flat_Pack_Mode
OR Demo_Mode  ; With or without trays
ANDLD
ORLD
ORLD
NOT(520)
OUT opState_V5B_Slow_Top_Vent  ; V5B Slow Top Vent TEST

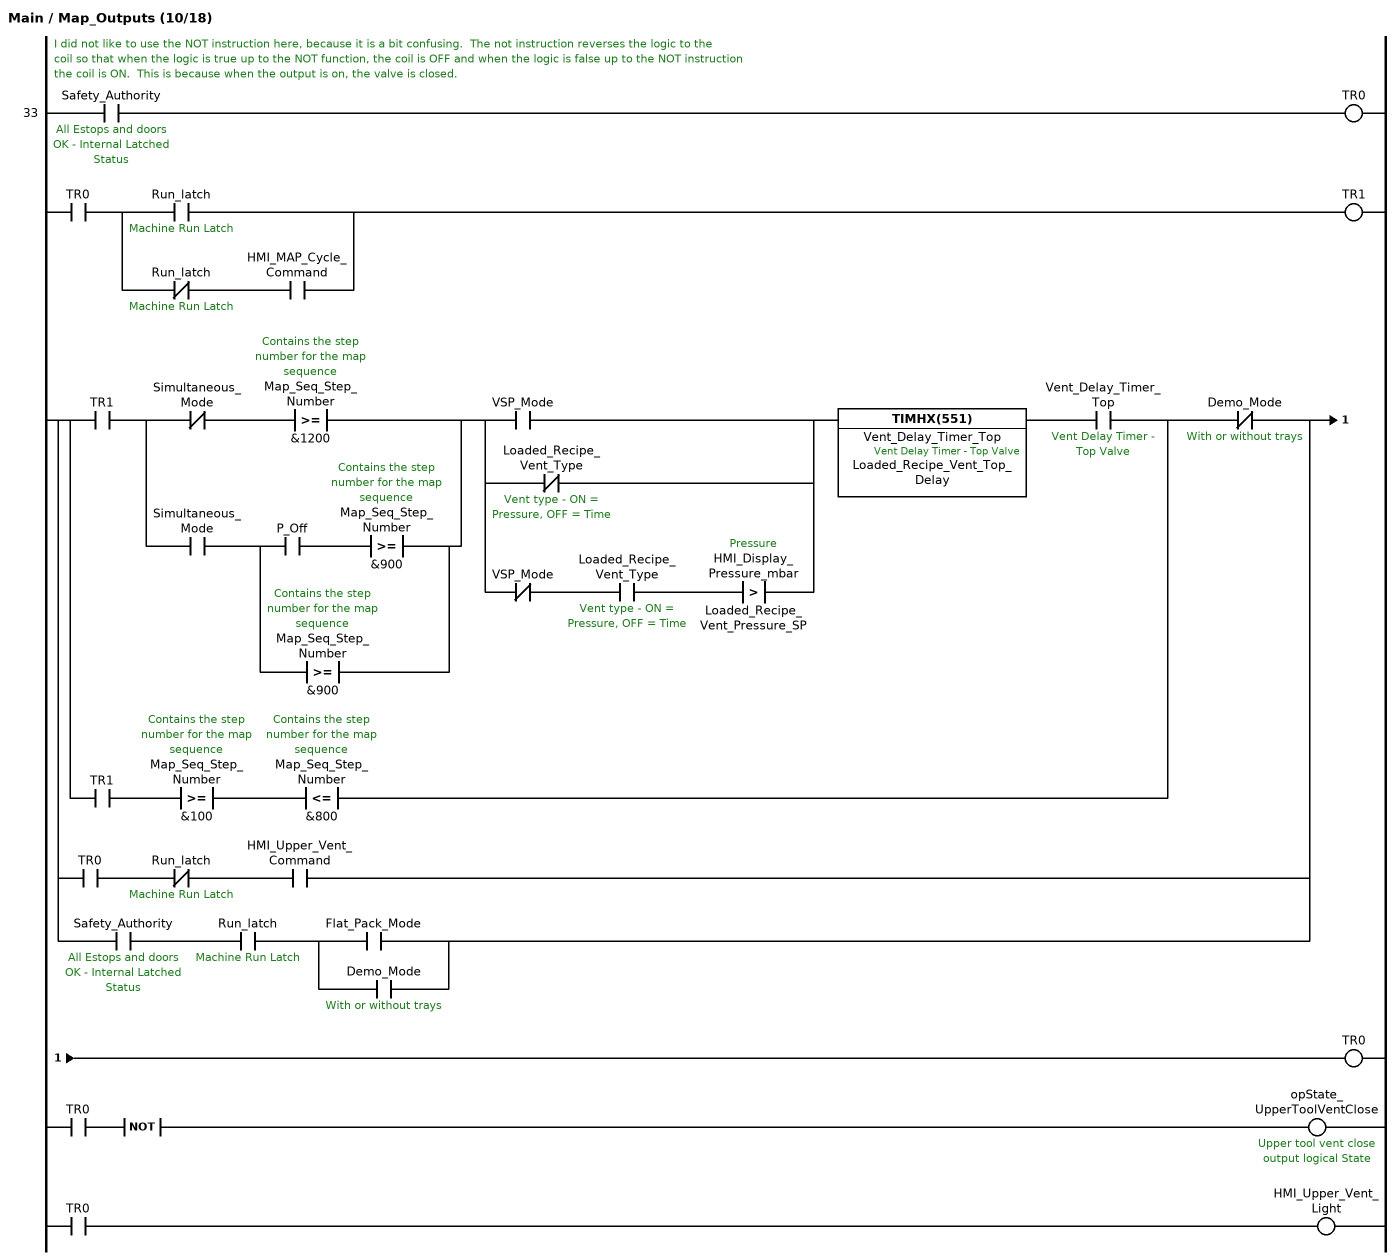
; rung 33: I did not like to use the NOT instruction here, because it is a bit confusing.  The not instruction reverses the logic to the / coil so that when the logic is true up to the NOT function, the coil is OFF and when the logic is false up to the NOT instruction / the coil is ON.  This is because when the output is on, the valve is closed.
LD Safety_Authority  ; All Estops and doors OK - Internal Latched Status
OUT TR0
LD Run_latch  ; Machine Run Latch
LDNOT Run_latch  ; Machine Run Latch
AND HMI_MAP_Cycle_Command
ORLD
ANDLD
OUT TR1
LDNOT Simultaneous_Mode
AND>=(325) Map_Seq_Step_Number &1200  ; Contains the step number for the map sequence
LD Simultaneous_Mode
LD P_Off
AND>=(325) Map_Seq_Step_Number &900  ; Contains the step number for the map sequence
OR>=(325) Map_Seq_Step_Number &900  ; Contains the step number for the map sequence
ANDLD
ORLD
ANDLD
LD VSP_Mode
ORNOT Loaded_Recipe_Vent_Type  ; Vent type - ON = Pressure, OFF = Time
LDNOT VSP_Mode
AND Loaded_Recipe_Vent_Type  ; Vent type - ON = Pressure, OFF = Time
AND>(320) HMI_Display_Pressure_mbar Loaded_Recipe_Vent_Pressure_SP  ; Pressure
ORLD
ANDLD
TIMHX(551) Vent_Delay_Timer_Top Loaded_Recipe_Vent_Top_Delay  ; Vent Delay Timer - Top Valve
AND Vent_Delay_Timer_Top  ; Vent Delay Timer - Top Valve
LD TR1
AND>=(325) Map_Seq_Step_Number &100  ; Contains the step number for the map sequence
AND<=(315) Map_Seq_Step_Number &800  ; Contains the step number for the map sequence
ORLD
ANDNOT Demo_Mode  ; With or without trays
LD TR0
ANDNOT Run_latch  ; Machine Run Latch
AND HMI_Upper_Vent_Command
LD Safety_Authority  ; All Estops and doors OK - Internal Latched Status
AND Run_latch  ; Machine Run Latch
LD Flat_Pack_Mode
OR Demo_Mode  ; With or without trays
ANDLD
ORLD
ORLD
OUT TR0
NOT(520)
OUT opState_UpperToolVentClose  ; Upper tool vent close output logical State
LD TR0
OUT HMI_Upper_Vent_Light

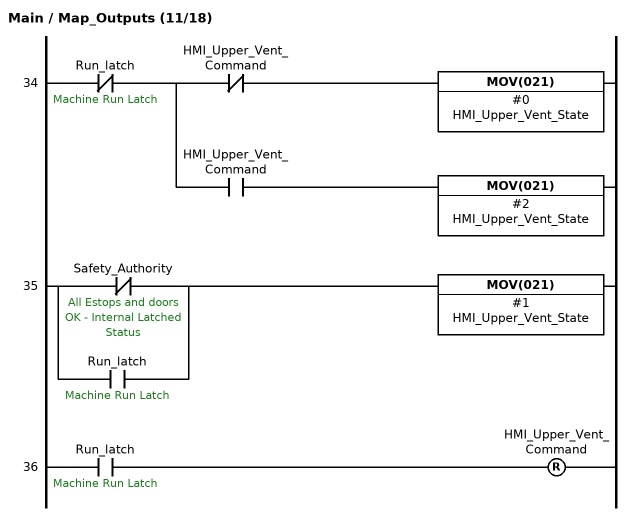
; rung 34
LDNOT Run_latch  ; Machine Run Latch
OUT TR0
ANDNOT HMI_Upper_Vent_Command
MOV(021) #0 HMI_Upper_Vent_State
LD TR0
AND HMI_Upper_Vent_Command
MOV(021) #2 HMI_Upper_Vent_State
; rung 35
LDNOT Safety_Authority  ; All Estops and doors OK - Internal Latched Status
OR Run_latch  ; Machine Run Latch
MOV(021) #1 HMI_Upper_Vent_State
; rung 36
LD Run_latch  ; Machine Run Latch
RSET HMI_Upper_Vent_Command

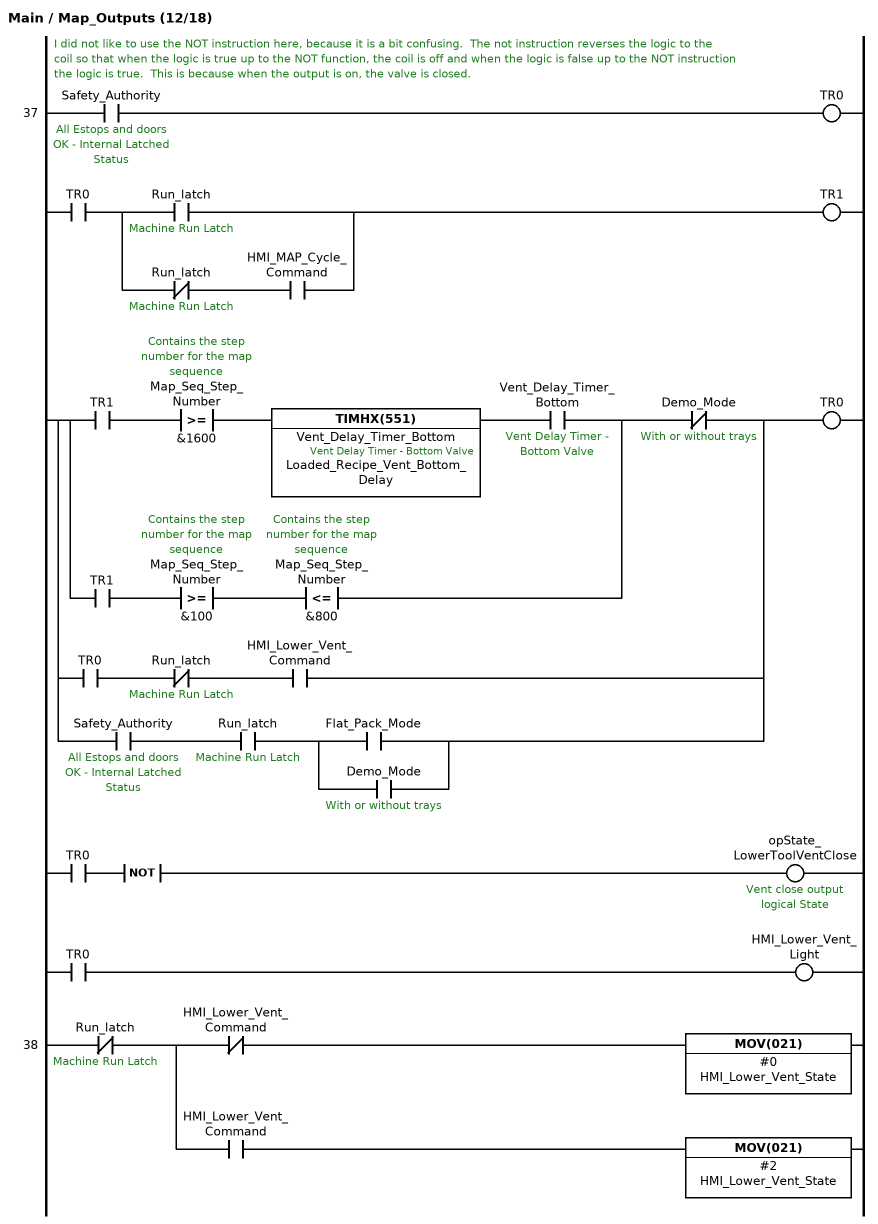
; rung 37: I did not like to use the NOT instruction here, because it is a bit confusing.  The not instruction reverses the logic to the / coil so that when the logic is true up to the NOT function, the coil is off and when the logic is false up to the NOT instruction / the logic is true.  This is because when the output is on, the valve is closed.
LD Safety_Authority  ; All Estops and doors OK - Internal Latched Status
OUT TR0
LD Run_latch  ; Machine Run Latch
LDNOT Run_latch  ; Machine Run Latch
AND HMI_MAP_Cycle_Command
ORLD
ANDLD
OUT TR1
AND>=(325) Map_Seq_Step_Number &1600  ; Contains the step number for the map sequence
TIMHX(551) Vent_Delay_Timer_Bottom Loaded_Recipe_Vent_Bottom_Delay  ; Vent Delay Timer - Bottom Valve
AND Vent_Delay_Timer_Bottom  ; Vent Delay Timer - Bottom Valve
LD TR1
AND>=(325) Map_Seq_Step_Number &100  ; Contains the step number for the map sequence
AND<=(315) Map_Seq_Step_Number &800  ; Contains the step number for the map sequence
ORLD
ANDNOT Demo_Mode  ; With or without trays
LD TR0
ANDNOT Run_latch  ; Machine Run Latch
AND HMI_Lower_Vent_Command
LD Safety_Authority  ; All Estops and doors OK - Internal Latched Status
AND Run_latch  ; Machine Run Latch
LD Flat_Pack_Mode
OR Demo_Mode  ; With or without trays
ANDLD
ORLD
ORLD
OUT TR0
NOT(520)
OUT opState_LowerToolVentClose  ; Vent close output logical State
LD TR0
OUT HMI_Lower_Vent_Light
; rung 38
LDNOT Run_latch  ; Machine Run Latch
OUT TR0
ANDNOT HMI_Lower_Vent_Command
MOV(021) #0 HMI_Lower_Vent_State
LD TR0
AND HMI_Lower_Vent_Command
MOV(021) #2 HMI_Lower_Vent_State

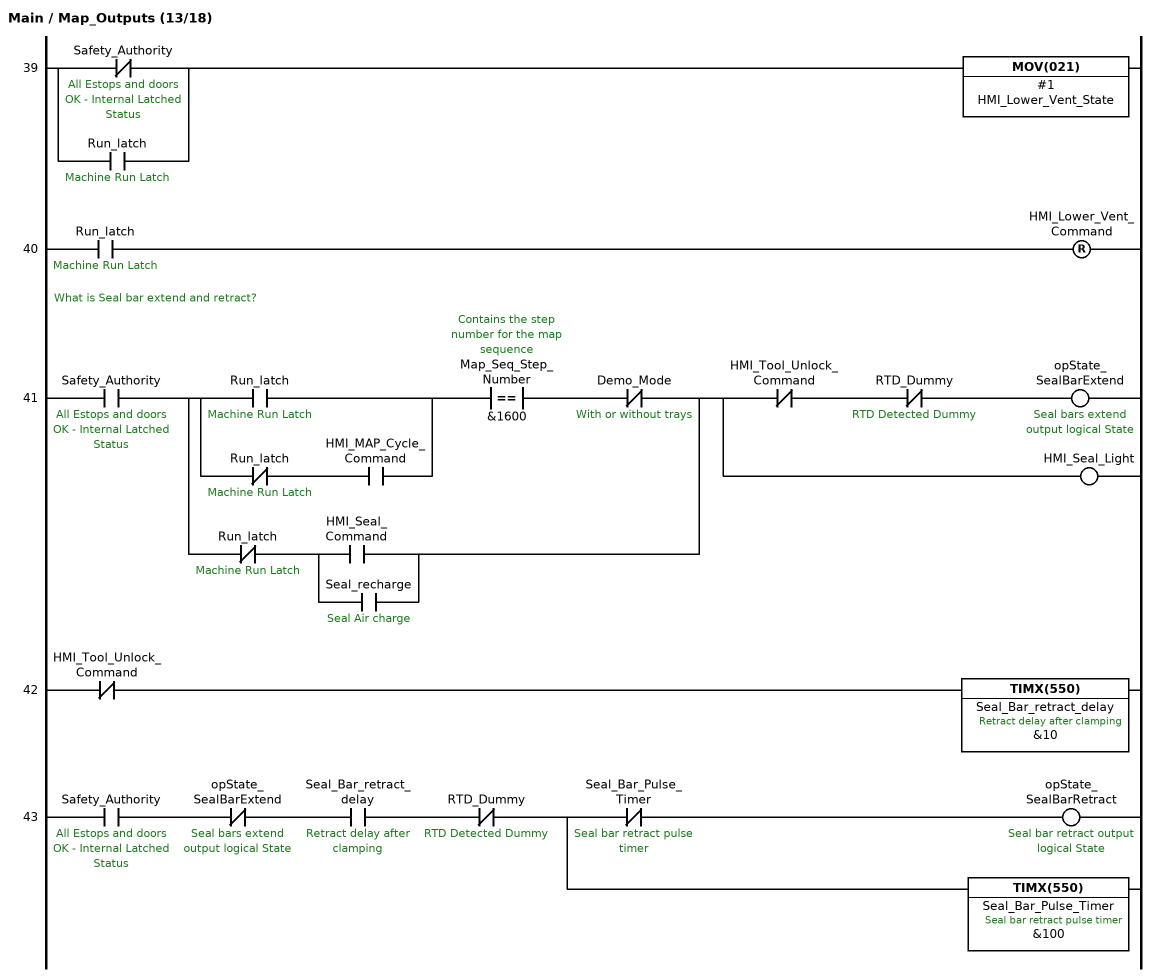
; rung 39
LDNOT Safety_Authority  ; All Estops and doors OK - Internal Latched Status
OR Run_latch  ; Machine Run Latch
MOV(021) #1 HMI_Lower_Vent_State
; rung 40
LD Run_latch  ; Machine Run Latch
RSET HMI_Lower_Vent_Command
; rung 41: What is Seal bar extend and retract?
LD Safety_Authority  ; All Estops and doors OK - Internal Latched Status
LD Run_latch  ; Machine Run Latch
LDNOT Run_latch  ; Machine Run Latch
AND HMI_MAP_Cycle_Command
ORLD
AND=(300) Map_Seq_Step_Number &1600  ; Contains the step number for the map sequence
ANDNOT Demo_Mode  ; With or without trays
LDNOT Run_latch  ; Machine Run Latch
LD HMI_Seal_Command
OR Seal_recharge  ; Seal Air charge
ANDLD
ORLD
ANDLD
OUT TR0
ANDNOT HMI_Tool_Unlock_Command
ANDNOT RTD_Dummy  ; RTD Detected Dummy
OUT opState_SealBarExtend  ; Seal bars extend output logical State
LD TR0
OUT HMI_Seal_Light
; rung 42
LDNOT HMI_Tool_Unlock_Command
TIMX(550) Seal_Bar_retract_delay &10  ; Retract delay after clamping
; rung 43
LD Safety_Authority  ; All Estops and doors OK - Internal Latched Status
ANDNOT opState_SealBarExtend  ; Seal bars extend output logical State
AND Seal_Bar_retract_delay  ; Retract delay after clamping
ANDNOT RTD_Dummy  ; RTD Detected Dummy
OUT TR0
ANDNOT Seal_Bar_Pulse_Timer  ; Seal bar retract pulse timer
OUT opState_SealBarRetract  ; Seal bar retract output logical State
LD TR0
TIMX(550) Seal_Bar_Pulse_Timer &100  ; Seal bar retract pulse timer

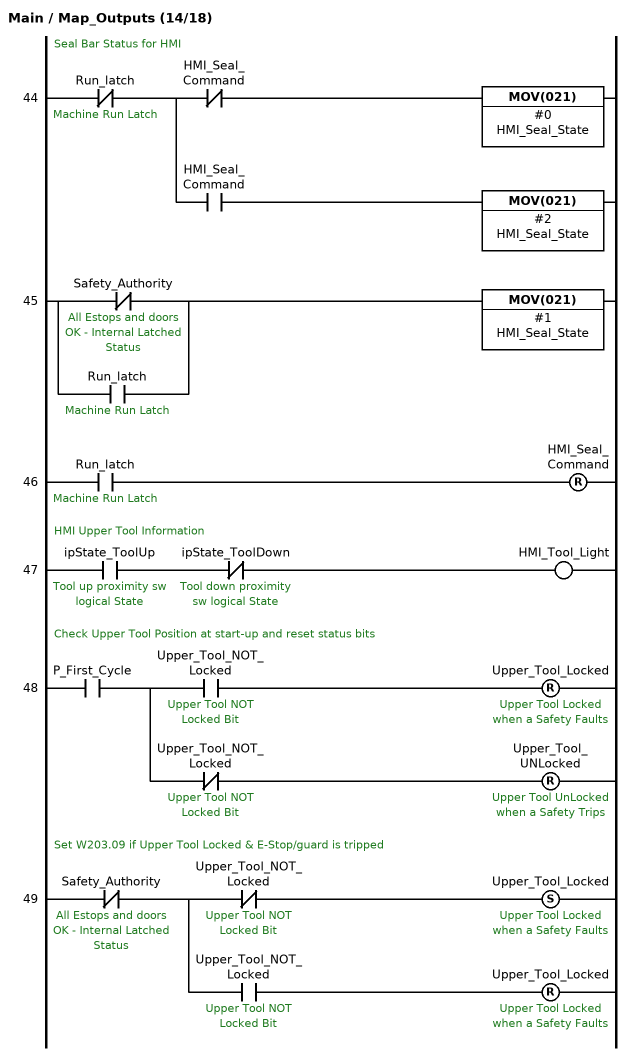
; rung 44: Seal Bar Status for HMI
LDNOT Run_latch  ; Machine Run Latch
OUT TR0
ANDNOT HMI_Seal_Command
MOV(021) #0 HMI_Seal_State
LD TR0
AND HMI_Seal_Command
MOV(021) #2 HMI_Seal_State
; rung 45
LDNOT Safety_Authority  ; All Estops and doors OK - Internal Latched Status
OR Run_latch  ; Machine Run Latch
MOV(021) #1 HMI_Seal_State
; rung 46
LD Run_latch  ; Machine Run Latch
RSET HMI_Seal_Command
; rung 47: HMI Upper Tool Information
LD ipState_ToolUp  ; Tool up proximity sw logical State
ANDNOT ipState_ToolDown  ; Tool down proximity sw logical State
OUT HMI_Tool_Light
; rung 48: Check Upper Tool Position at start-up and reset status bits
LD P_First_Cycle
OUT TR0
AND Upper_Tool_NOT_Locked  ; Upper Tool NOT Locked Bit
RSET Upper_Tool_Locked  ; Upper Tool Locked when a Safety Faults
LD TR0
ANDNOT Upper_Tool_NOT_Locked  ; Upper Tool NOT Locked Bit
RSET Upper_Tool_UNLocked  ; Upper Tool UnLocked when a Safety Trips
; rung 49: Set W203.09 if Upper Tool Locked & E-Stop/guard is tripped
LDNOT Safety_Authority  ; All Estops and doors OK - Internal Latched Status
OUT TR0
ANDNOT Upper_Tool_NOT_Locked  ; Upper Tool NOT Locked Bit
SET Upper_Tool_Locked  ; Upper Tool Locked when a Safety Faults
LD TR0
AND Upper_Tool_NOT_Locked  ; Upper Tool NOT Locked Bit
RSET Upper_Tool_Locked  ; Upper Tool Locked when a Safety Faults

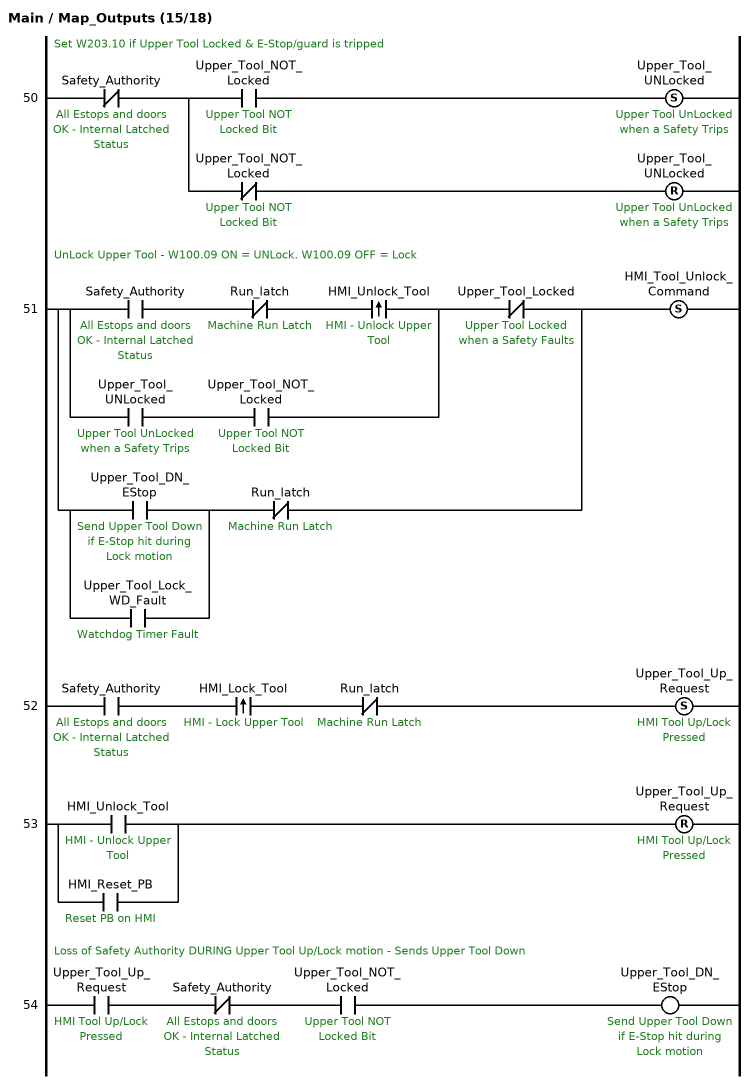
; rung 50: Set W203.10 if Upper Tool Locked & E-Stop/guard is tripped
LDNOT Safety_Authority  ; All Estops and doors OK - Internal Latched Status
OUT TR0
AND Upper_Tool_NOT_Locked  ; Upper Tool NOT Locked Bit
SET Upper_Tool_UNLocked  ; Upper Tool UnLocked when a Safety Trips
LD TR0
ANDNOT Upper_Tool_NOT_Locked  ; Upper Tool NOT Locked Bit
RSET Upper_Tool_UNLocked  ; Upper Tool UnLocked when a Safety Trips
; rung 51: UnLock Upper Tool - W100.09 ON = UNLock. W100.09 OFF = Lock
LD Safety_Authority  ; All Estops and doors OK - Internal Latched Status
ANDNOT Run_latch  ; Machine Run Latch
@AND HMI_Unlock_Tool  ; HMI - Unlock Upper Tool
LD Upper_Tool_UNLocked  ; Upper Tool UnLocked when a Safety Trips
AND Upper_Tool_NOT_Locked  ; Upper Tool NOT Locked Bit
ORLD
ANDNOT Upper_Tool_Locked  ; Upper Tool Locked when a Safety Faults
LD Upper_Tool_DN_EStop  ; Send Upper Tool Down if E-Stop hit during Lock motion
OR Upper_Tool_Lock_WD_Fault  ; Watchdog Timer Fault
ANDNOT Run_latch  ; Machine Run Latch
ORLD
SET HMI_Tool_Unlock_Command
; rung 52
LD Safety_Authority  ; All Estops and doors OK - Internal Latched Status
@AND HMI_Lock_Tool  ; HMI - Lock Upper Tool
ANDNOT Run_latch  ; Machine Run Latch
SET Upper_Tool_Up_Request  ; HMI Tool Up/Lock Pressed
; rung 53
LD HMI_Unlock_Tool  ; HMI - Unlock Upper Tool
OR HMI_Reset_PB  ; Reset PB on HMI
RSET Upper_Tool_Up_Request  ; HMI Tool Up/Lock Pressed
; rung 54: Loss of Safety Authority DURING Upper Tool Up/Lock motion - Sends Upper Tool Down
LD Upper_Tool_Up_Request  ; HMI Tool Up/Lock Pressed
ANDNOT Safety_Authority  ; All Estops and doors OK - Internal Latched Status
AND Upper_Tool_NOT_Locked  ; Upper Tool NOT Locked Bit
OUT Upper_Tool_DN_EStop  ; Send Upper Tool Down if E-Stop hit during Lock motion

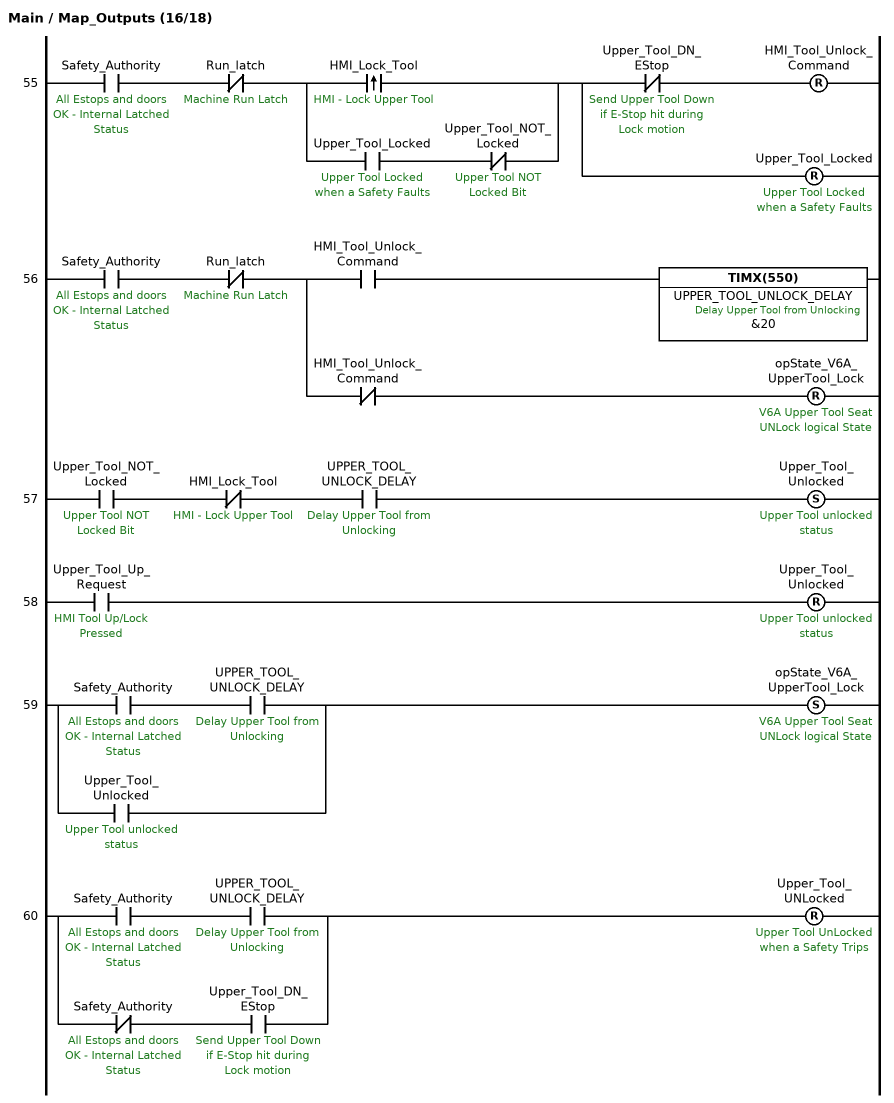
; rung 55
LD Safety_Authority  ; All Estops and doors OK - Internal Latched Status
ANDNOT Run_latch  ; Machine Run Latch
@LD HMI_Lock_Tool  ; HMI - Lock Upper Tool
LD Upper_Tool_Locked  ; Upper Tool Locked when a Safety Faults
ANDNOT Upper_Tool_NOT_Locked  ; Upper Tool NOT Locked Bit
ORLD
ANDLD
OUT TR0
ANDNOT Upper_Tool_DN_EStop  ; Send Upper Tool Down if E-Stop hit during Lock motion
RSET HMI_Tool_Unlock_Command
LD TR0
RSET Upper_Tool_Locked  ; Upper Tool Locked when a Safety Faults
; rung 56
LD Safety_Authority  ; All Estops and doors OK - Internal Latched Status
ANDNOT Run_latch  ; Machine Run Latch
OUT TR0
AND HMI_Tool_Unlock_Command
TIMX(550) UPPER_TOOL_UNLOCK_DELAY &20  ; Delay Upper Tool from Unlocking
LD TR0
ANDNOT HMI_Tool_Unlock_Command
RSET opState_V6A_UpperTool_Lock  ; V6A Upper Tool Seat UNLock logical State
; rung 57
LD Upper_Tool_NOT_Locked  ; Upper Tool NOT Locked Bit
ANDNOT HMI_Lock_Tool  ; HMI - Lock Upper Tool
AND UPPER_TOOL_UNLOCK_DELAY  ; Delay Upper Tool from Unlocking
SET Upper_Tool_Unlocked  ; Upper Tool unlocked status
; rung 58
LD Upper_Tool_Up_Request  ; HMI Tool Up/Lock Pressed
RSET Upper_Tool_Unlocked  ; Upper Tool unlocked status
; rung 59
LD Safety_Authority  ; All Estops and doors OK - Internal Latched Status
AND UPPER_TOOL_UNLOCK_DELAY  ; Delay Upper Tool from Unlocking
OR Upper_Tool_Unlocked  ; Upper Tool unlocked status
SET opState_V6A_UpperTool_Lock  ; V6A Upper Tool Seat UNLock logical State
; rung 60
LD Safety_Authority  ; All Estops and doors OK - Internal Latched Status
AND UPPER_TOOL_UNLOCK_DELAY  ; Delay Upper Tool from Unlocking
LDNOT Safety_Authority  ; All Estops and doors OK - Internal Latched Status
AND Upper_Tool_DN_EStop  ; Send Upper Tool Down if E-Stop hit during Lock motion
ORLD
RSET Upper_Tool_UNLocked  ; Upper Tool UnLocked when a Safety Trips

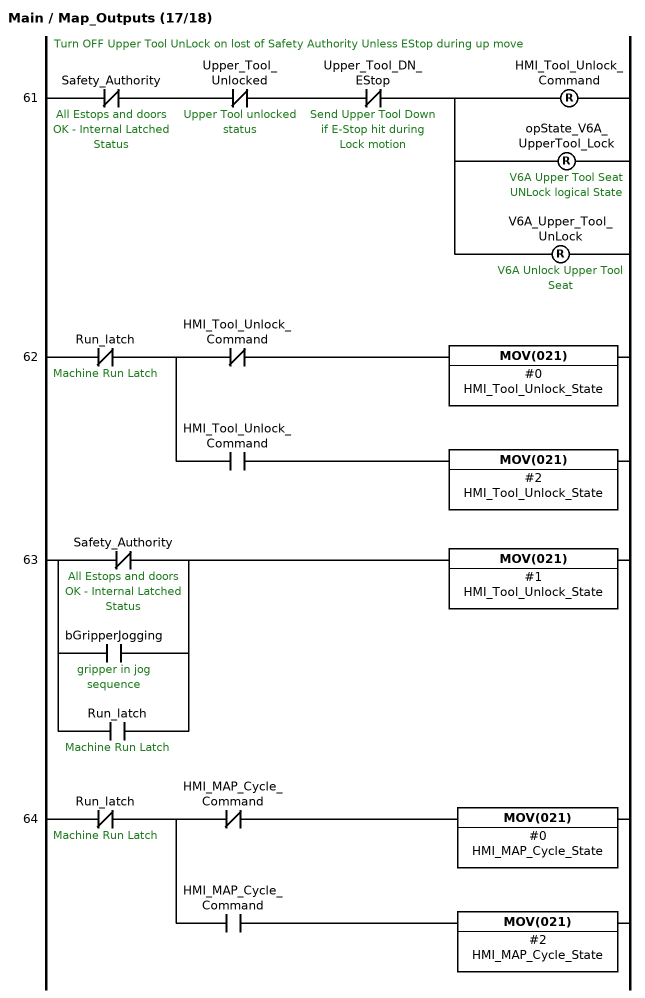
; rung 61: Turn OFF Upper Tool UnLock on lost of Safety Authority Unless EStop during up move
LDNOT Safety_Authority  ; All Estops and doors OK - Internal Latched Status
ANDNOT Upper_Tool_Unlocked  ; Upper Tool unlocked status
ANDNOT Upper_Tool_DN_EStop  ; Send Upper Tool Down if E-Stop hit during Lock motion
RSET HMI_Tool_Unlock_Command
RSET opState_V6A_UpperTool_Lock  ; V6A Upper Tool Seat UNLock logical State
RSET V6A_Upper_Tool_UnLock  ; V6A Unlock Upper Tool Seat
; rung 62
LDNOT Run_latch  ; Machine Run Latch
OUT TR0
ANDNOT HMI_Tool_Unlock_Command
MOV(021) #0 HMI_Tool_Unlock_State
LD TR0
AND HMI_Tool_Unlock_Command
MOV(021) #2 HMI_Tool_Unlock_State
; rung 63
LDNOT Safety_Authority  ; All Estops and doors OK - Internal Latched Status
OR bGripperJogging  ; gripper in jog sequence
OR Run_latch  ; Machine Run Latch
MOV(021) #1 HMI_Tool_Unlock_State
; rung 64
LDNOT Run_latch  ; Machine Run Latch
OUT TR0
ANDNOT HMI_MAP_Cycle_Command
MOV(021) #0 HMI_MAP_Cycle_State
LD TR0
AND HMI_MAP_Cycle_Command
MOV(021) #2 HMI_MAP_Cycle_State

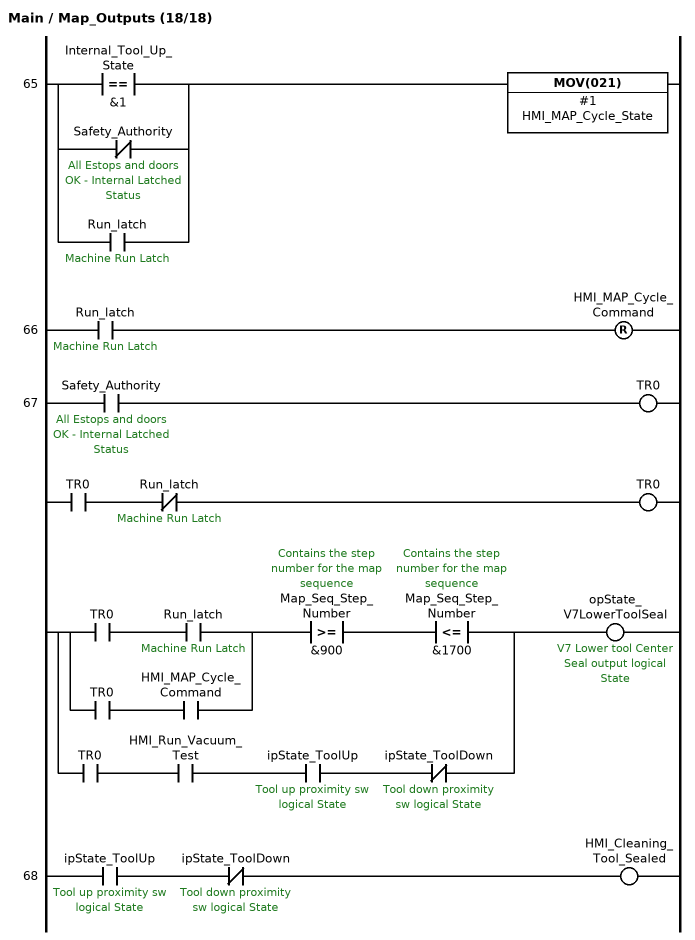
; rung 65
LD=(300) Internal_Tool_Up_State &1
ORNOT Safety_Authority  ; All Estops and doors OK - Internal Latched Status
OR Run_latch  ; Machine Run Latch
MOV(021) #1 HMI_MAP_Cycle_State
; rung 66
LD Run_latch  ; Machine Run Latch
RSET HMI_MAP_Cycle_Command
; rung 67
LD Safety_Authority  ; All Estops and doors OK - Internal Latched Status
OUT TR0
AND Run_latch  ; Machine Run Latch
LD TR0
ANDNOT Run_latch  ; Machine Run Latch
OUT TR0
AND HMI_MAP_Cycle_Command
ORLD
AND>=(325) Map_Seq_Step_Number &900  ; Contains the step number for the map sequence
AND<=(315) Map_Seq_Step_Number &1700  ; Contains the step number for the map sequence
LD TR0
AND HMI_Run_Vacuum_Test
AND ipState_ToolUp  ; Tool up proximity sw logical State
ANDNOT ipState_ToolDown  ; Tool down proximity sw logical State
ORLD
OUT opState_V7LowerToolSeal  ; V7 Lower tool Center Seal output logical State
; rung 68
LD ipState_ToolUp  ; Tool up proximity sw logical State
ANDNOT ipState_ToolDown  ; Tool down proximity sw logical State
OUT HMI_Cleaning_Tool_Sealed

### Section Film_control

